//     Standard Inputs/Fix01.N22/I <-> Channel 1/Input
//     Standard Inputs/Fix01.N22/I @bit 1 <-> Channel 2/Input
//     Standard Inputs/Fix01.N22/I @bit 2 <-> Channel 3/Input
//     Standard Inputs/Fix01.N22/I @bit 3 <-> Channel 4/Input
//     Standard Inputs/Fix01.N22/I @bit 4 <-> Channel 5/Input
//     Standard Inputs/Fix01.N22/I @bit 5 <-> Channel 6/Input
//     Standard Inputs/Fix01.N22/I @bit 6 <-> Channel 7/Input
//     Standard Inputs/Fix01.N22/I @bit 7 <-> Channel 8/Input
//     Standard Inputs/Fix01.N22/InfoData/State <-> InfoData/State
//     Standard Inputs/Fix01.N22/Wc_State <-> WcState/WcState
//   SODG11_SSCC610_2403701_PLC/SODG11_SSCC610_2403701_PLC Instance <-> EtherCAT Master (EtherCAT)/IC01.T01 (EK1100)/IC01.T16 (EK1122)/Fix01.N23 (EP1008-0002)
//     Standard Inputs/Fix01.N23/I <-> Channel 1/Input
//     Standard Inputs/Fix01.N23/I @bit 1 <-> Channel 2/Input
//     Standard Inputs/Fix01.N23/I @bit 2 <-> Channel 3/Input
//     Standard Inputs/Fix01.N23/I @bit 3 <-> Channel 4/Input
//     Standard Inputs/Fix01.N23/I @bit 4 <-> Channel 5/Input
//     Standard Inputs/Fix01.N23/I @bit 5 <-> Channel 6/Input
//     Standard Inputs/Fix01.N23/I @bit 6 <-> Channel 7/Input
//     Standard Inputs/Fix01.N23/I @bit 7 <-> Channel 8/Input
//     Standard Inputs/Fix01.N23/InfoData/State <-> InfoData/State
//     Standard Inputs/Fix01.N23/Wc_State <-> WcState/WcState
//   SODG11_SSCC610_2403701_PLC/SODG11_SSCC610_2403701_PLC Instance <-> EtherCAT Master (EtherCAT)/IC01.T01 (EK1100)/IC01.T16 (EK1122)/Fix01.N24 (EP1008-0002)
//     Standard Inputs/Fix01.N24/I <-> Channel 1/Input
//     Standard Inputs/Fix01.N24/I @bit 1 <-> Channel 2/Input
//     Standard Inputs/Fix01.N24/I @bit 2 <-> Channel 3/Input
//     Standard Inputs/Fix01.N24/I @bit 3 <-> Channel 4/Input
//     Standard Inputs/Fix01.N24/I @bit 4 <-> Channel 5/Input
//     Standard Inputs/Fix01.N24/I @bit 5 <-> Channel 6/Input
//     Standard Inputs/Fix01.N24/I @bit 6 <-> Channel 7/Input
//     Standard Inputs/Fix01.N24/I @bit 7 <-> Channel 8/Input
//     Standard Inputs/Fix01.N24/InfoData/State <-> InfoData/State
//     Standard Inputs/Fix01.N24/Wc_State <-> WcState/WcState
//   SODG11_SSCC610_2403701_PLC/SODG11_SSCC610_2403701_PLC Instance <-> EtherCAT Master (EtherCAT)/IC01.T01 (EK1100)/IC01.T16 (EK1122)/Fix01.N25 (EP1008-0002)
//     Standard Inputs/Fix01.N25/I <-> Channel 1/Input
//     Standard Inputs/Fix01.N25/I @bit 1 <-> Channel 2/Input
//     Standard Inputs/Fix01.N25/I @bit 2 <-> Channel 3/Input
//     Standard Inputs/Fix01.N25/I @bit 3 <-> Channel 4/Input
//     Standard Inputs/Fix01.N25/I @bit 4 <-> Channel 5/Input
//     Standard Inputs/Fix01.N25/I @bit 5 <-> Channel 6/Input
//     Standard Inputs/Fix01.N25/I @bit 6 <-> Channel 7/Input
//     Standard Inputs/Fix01.N25/I @bit 7 <-> Channel 8/Input
//     Standard Inputs/Fix01.N25/InfoData/State <-> InfoData/State
//     Standard Inputs/Fix01.N25/Wc_State <-> WcState/WcState
//   SODG11_SSCC610_2403701_PLC/SODG11_SSCC610_2403701_PLC Instance <-> EtherCAT Master (EtherCAT)/IC01.T01 (EK1100)/IC01.T16 (EK1122)/Fix01.N26 (EP1008-0002)
//     Standard Inputs/Fix01.N26/I <-> Channel 1/Input
//     Standard Inputs/Fix01.N26/I @bit 1 <-> Channel 2/Input
//     Standard Inputs/Fix01.N26/I @bit 2 <-> Channel 3/Input
//     Standard Inputs/Fix01.N26/I @bit 3 <-> Channel 4/Input
//     Standard Inputs/Fix01.N26/I @bit 4 <-> Channel 5/Input
//     Standard Inputs/Fix01.N26/I @bit 5 <-> Channel 6/Input
//     Standard Inputs/Fix01.N26/I @bit 6 <-> Channel 7/Input
//     Standard Inputs/Fix01.N26/I @bit 7 <-> Channel 8/Input
//     Standard Inputs/Fix01.N26/InfoData/State <-> InfoData/State
//     Standard Inputs/Fix01.N26/Wc_State <-> WcState/WcState
//   SODG11_SSCC610_2403701_PLC/SODG11_SSCC610_2403701_PLC Instance <-> EtherCAT Master (EtherCAT)/IC01.T01 (EK1100)/IC01.T16 (EK1122)/Fix01.N27 (EP1008-0002)
//     Standard Inputs/Fix01.N27/I <-> Channel 1/Input
//     Standard Inputs/Fix01.N27/I @bit 1 <-> Channel 2/Input
//     Standard Inputs/Fix01.N27/I @bit 2 <-> Channel 3/Input
//     Standard Inputs/Fix01.N27/I @bit 3 <-> Channel 4/Input
//     Standard Inputs/Fix01.N27/I @bit 4 <-> Channel 5/Input
//     Standard Inputs/Fix01.N27/I @bit 5 <-> Channel 6/Input
//     Standard Inputs/Fix01.N27/I @bit 6 <-> Channel 7/Input
//     Standard Inputs/Fix01.N27/I @bit 7 <-> Channel 8/Input
//     Standard Inputs/Fix01.N27/InfoData/State <-> InfoData/State
//     Standard Inputs/Fix01.N27/Wc_State <-> WcState/WcState
//   SODG11_SSCC610_2403701_PLC/SODG11_SSCC610_2403701_PLC Instance <-> EtherCAT Master (EtherCAT)/IC01.T01 (EK1100)/IC01.T16 (EK1122)/Fix01.N28 (EP1008-0002)
//     Standard Inputs/Fix01.N28/I <-> Channel 1/Input
//     Standard Inputs/Fix01.N28/I @bit 1 <-> Channel 2/Input
//     Standard Inputs/Fix01.N28/I @bit 2 <-> Channel 3/Input
//     Standard Inputs/Fix01.N28/I @bit 3 <-> Channel 4/Input
//     Standard Inputs/Fix01.N28/I @bit 4 <-> Channel 5/Input
//     Standard Inputs/Fix01.N28/I @bit 5 <-> Channel 6/Input
//     Standard Inputs/Fix01.N28/I @bit 6 <-> Channel 7/Input
//     Standard Inputs/Fix01.N28/I @bit 7 <-> Channel 8/Input
//     Standard Inputs/Fix01.N28/InfoData/State <-> InfoData/State
//     Standard Inputs/Fix01.N28/Wc_State <-> WcState/WcState
//   SODG11_SSCC610_2403701_PLC/SODG11_SSCC610_2403701_PLC Instance <-> EtherCAT Master (EtherCAT)/IC01.T01 (EK1100)/IC01.T16 (EK1122)/Fix01.N29 (EP1008-0002)
//     Standard Inputs/Fix01.N29/I <-> Channel 1/Input
//     Standard Inputs/Fix01.N29/I @bit 1 <-> Channel 2/Input
//     Standard Inputs/Fix01.N29/I @bit 2 <-> Channel 3/Input
//     Standard Inputs/Fix01.N29/I @bit 3 <-> Channel 4/Input
//     Standard Inputs/Fix01.N29/I @bit 4 <-> Channel 5/Input
//     Standard Inputs/Fix01.N29/I @bit 5 <-> Channel 6/Input
//     Standard Inputs/Fix01.N29/I @bit 6 <-> Channel 7/Input
//     Standard Inputs/Fix01.N29/I @bit 7 <-> Channel 8/Input
//     Standard Inputs/Fix01.N29/InfoData/State <-> InfoData/State
//     Standard Inputs/Fix01.N29/Wc_State <-> WcState/WcState
//   SODG11_SSCC610_2403701_PLC/SODG11_SSCC610_2403701_PLC Instance <-> EtherCAT Master (EtherCAT)/IC01.T01 (EK1100)/IC01.T16 (EK1122)/Fix01.N30 (EP1008-0002)
//     Standard Inputs/Fix01.N30/I <-> Channel 1/Input
//     Standard Inputs/Fix01.N30/I @bit 1 <-> Channel 2/Input
//     Standard Inputs/Fix01.N30/I @bit 2 <-> Channel 3/Input
//     Standard Inputs/Fix01.N30/I @bit 3 <-> Channel 4/Input
//     Standard Inputs/Fix01.N30/I @bit 4 <-> Channel 5/Input
//     Standard Inputs/Fix01.N30/I @bit 5 <-> Channel 6/Input
//     Standard Inputs/Fix01.N30/I @bit 6 <-> Channel 7/Input
//     Standard Inputs/Fix01.N30/I @bit 7 <-> Channel 8/Input
//     Standard Inputs/Fix01.N30/InfoData/State <-> InfoData/State
//     Standard Inputs/Fix01.N30/Wc_State <-> WcState/WcState
//   SODG11_SSCC610_2403701_PLC/SODG11_SSCC610_2403701_PLC Instance <-> EtherCAT Master (EtherCAT)/IC01.T01 (EK1100)/IC01.T16 (EK1122)/Fix01.N31 (EP1008-0002)
//     Standard Inputs/Fix01.N31/I <-> Channel 1/Input
//     Standard Inputs/Fix01.N31/I @bit 1 <-> Channel 2/Input
//     Standard Inputs/Fix01.N31/I @bit 2 <-> Channel 3/Input
//     Standard Inputs/Fix01.N31/I @bit 3 <-> Channel 4/Input
//     Standard Inputs/Fix01.N31/I @bit 4 <-> Channel 5/Input
//     Standard Inputs/Fix01.N31/I @bit 5 <-> Channel 6/Input
//     Standard Inputs/Fix01.N31/I @bit 6 <-> Channel 7/Input
//     Standard Inputs/Fix01.N31/I @bit 7 <-> Channel 8/Input
//     Standard Inputs/Fix01.N31/InfoData/State <-> InfoData/State
//     Standard Inputs/Fix01.N31/Wc_State <-> WcState/WcState
//   SODG11_SSCC610_2403701_PLC/SODG11_SSCC610_2403701_PLC Instance <-> EtherCAT Master (EtherCAT)/IC01.T01 (EK1100)/IC01.T16 (EK1122)/Fix01.N90 (EP9214-0023)
//     Standard Inputs/Fix01.N90_STAT/Channel_1/Channel_Error <-> DPO Inputs Channel 1/Channel Error
//     Standard Inputs/Fix01.N90_STAT/Channel_2/Channel_Error <-> DPO Inputs Channel 2/Channel Error
//     Standard Inputs/Fix01.N90_STAT/Channel_3/Channel_Error <-> DPO Inputs Channel 3/Channel Error
//     Standard Inputs/Fix01.N90_STAT/Channel_4/Channel_Error <-> DPO Inputs Channel 4/Channel Error
//     Standard Inputs/Fix01.N90_STAT/Channel_1/Error_Up <-> DPO Inputs Channel 1/Error Up
//     Standard Inputs/Fix01.N90_STAT/Channel_2/Error_Up <-> DPO Inputs Channel 2/Error Up
//     Standard Inputs/Fix01.N90_STAT/Channel_3/Error_Up <-> DPO Inputs Channel 3/Error Up
//     Standard Inputs/Fix01.N90_STAT/Channel_4/Error_Up <-> DPO Inputs Channel 4/Error Up
//     Standard Inputs/Fix01.N90_STAT/Channel_1/Error_Us <-> DPO Inputs Channel 1/Error Us
//     Standard Inputs/Fix01.N90_STAT/Channel_2/Error_Us <-> DPO Inputs Channel 2/Error Us
//     Standard Inputs/Fix01.N90_STAT/Channel_3/Error_Us <-> DPO Inputs Channel 3/Error Us
//     Standard Inputs/Fix01.N90_STAT/Channel_4/Error_Us <-> DPO Inputs Channel 4/Error Us
//     Standard Inputs/Fix01.N90_STAT/Channel_1/Status_Up <-> DPO Inputs Channel 1/Status Up
//     Standard Inputs/Fix01.N90_STAT/Channel_2/Status_Up <-> DPO Inputs Channel 2/Status Up
//     Standard Inputs/Fix01.N90_STAT/Channel_3/Status_Up <-> DPO Inputs Channel 3/Status Up
//     Standard Inputs/Fix01.N90_STAT/Channel_4/Status_Up <-> DPO Inputs Channel 4/Status Up
//     Standard Inputs/Fix01.N90_STAT/Channel_1/Status_Us <-> DPO Inputs Channel 1/Status Us
//     Standard Inputs/Fix01.N90_STAT/Channel_2/Status_Us <-> DPO Inputs Channel 2/Status Us
//     Standard Inputs/Fix01.N90_STAT/Channel_3/Status_Us <-> DPO Inputs Channel 3/Status Us
//     Standard Inputs/Fix01.N90_STAT/Channel_4/Status_Us <-> DPO Inputs Channel 4/Status Us
//     Standard Inputs/Fix01.N90_STAT/Channel_1/SyncError <-> DPO Inputs Channel 1/Sync error
//     Standard Inputs/Fix01.N90_STAT/Channel_2/SyncError <-> DPO Inputs Channel 2/Sync error
//     Standard Inputs/Fix01.N90_STAT/Channel_3/SyncError <-> DPO Inputs Channel 3/Sync error
//     Standard Inputs/Fix01.N90_STAT/Channel_4/SyncError <-> DPO Inputs Channel 4/Sync error
//     Standard Inputs/Fix01.N90_STAT/Channel_1/TxPDO_State <-> DPO Inputs Channel 1/TxPDO State
//     Standard Inputs/Fix01.N90_STAT/Channel_2/TxPDO_State <-> DPO Inputs Channel 2/TxPDO State
//     Standard Inputs/Fix01.N90_STAT/Channel_3/TxPDO_State <-> DPO Inputs Channel 3/TxPDO State
//     Standard Inputs/Fix01.N90_STAT/Channel_4/TxPDO_State <-> DPO Inputs Channel 4/TxPDO State
//     Standard Inputs/Fix01.N90_STAT/Channel_1/TxPDO_Toggle <-> DPO Inputs Channel 1/TxPDO Toggle
//     Standard Inputs/Fix01.N90_STAT/Channel_2/TxPDO_Toggle <-> DPO Inputs Channel 2/TxPDO Toggle
//     Standard Inputs/Fix01.N90_STAT/Channel_3/TxPDO_Toggle <-> DPO Inputs Channel 3/TxPDO Toggle
//     Standard Inputs/Fix01.N90_STAT/Channel_4/TxPDO_Toggle <-> DPO Inputs Channel 4/TxPDO Toggle
//     Standard Inputs/Fix01.N90_STAT/Channel_1/Warning_Up <-> DPO Inputs Channel 1/Warning Up
//     Standard Inputs/Fix01.N90_STAT/Channel_2/Warning_Up <-> DPO Inputs Channel 2/Warning Up
//     Standard Inputs/Fix01.N90_STAT/Channel_3/Warning_Up <-> DPO Inputs Channel 3/Warning Up
//     Standard Inputs/Fix01.N90_STAT/Channel_4/Warning_Up <-> DPO Inputs Channel 4/Warning Up
//     Standard Inputs/Fix01.N90_STAT/Channel_1/Warning_Us <-> DPO Inputs Channel 1/Warning Us
//     Standard Inputs/Fix01.N90_STAT/Channel_2/Warning_Us <-> DPO Inputs Channel 2/Warning Us
//     Standard Inputs/Fix01.N90_STAT/Channel_3/Warning_Us <-> DPO Inputs Channel 3/Warning Us
//     Standard Inputs/Fix01.N90_STAT/Channel_4/Warning_Us <-> DPO Inputs Channel 4/Warning Us
//     Standard Inputs/Fix01.N90_STAT/Device/Global_Error_Bit <-> DPO Inputs Device/Global Error Bit
//     Standard Inputs/Fix01.N90_STAT/Device/Reset_Input <-> DPO Inputs Device/Reset Input
//     Standard Inputs/Fix01.N90_STAT/Device/Temperature_Error <-> DPO Inputs Device/Temperature Error
//     Standard Inputs/Fix01.N90_STAT/Device/Temperature_Warning <-> DPO Inputs Device/Temperature Warning
//     Standard Inputs/Fix01.N90_STAT/Device/TxPDO_State <-> DPO Inputs Device/TxPDO State
//     Standard Inputs/Fix01.N90_STAT/Device/TxPDO_Toggle <-> DPO Inputs Device/TxPDO Toggle
//     Standard Inputs/Fix01.N90_STAT/Device/Up_Error <-> DPO Inputs Device/Up Error
//     Standard Inputs/Fix01.N90_STAT/Device/Up_Warning <-> DPO Inputs Device/Up Warning
//     Standard Inputs/Fix01.N90_STAT/Device/Us_Error <-> DPO Inputs Device/Us Error
//     Standard Inputs/Fix01.N90_STAT/Device/Us_Warning <-> DPO Inputs Device/Us Warning
//     Standard Inputs/Fix01.N90_STAT/InfoData/AdsAddr <-> InfoData/AdsAddr
//     Standard Inputs/Fix01.N90_STAT/InfoData/State <-> InfoData/State
//     Standard Inputs/Fix01.N90_STAT/Wc_State <-> WcState/WcState
//     Standard Outputs/Fix01.N90_CMD/Channel1/Output_Up <-> DPO Outputs Channel 1/Output Up
//     Standard Outputs/Fix01.N90_CMD/Channel2/Output_Up <-> DPO Outputs Channel 2/Output Up
//     Standard Outputs/Fix01.N90_CMD/Channel3/Output_Up <-> DPO Outputs Channel 3/Output Up
//     Standard Outputs/Fix01.N90_CMD/Channel4/Output_Up <-> DPO Outputs Channel 4/Output Up
//     Standard Outputs/Fix01.N90_CMD/Channel1/Output_Us <-> DPO Outputs Channel 1/Output Us
//     Standard Outputs/Fix01.N90_CMD/Channel2/Output_Us <-> DPO Outputs Channel 2/Output Us
//     Standard Outputs/Fix01.N90_CMD/Channel3/Output_Us <-> DPO Outputs Channel 3/Output Us
//     Standard Outputs/Fix01.N90_CMD/Channel4/Output_Us <-> DPO Outputs Channel 4/Output Us
//     Standard Outputs/Fix01.N90_CMD/Channel1/Reset_Up <-> DPO Outputs Channel 1/Reset Up
//     Standard Outputs/Fix01.N90_CMD/Channel2/Reset_Up <-> DPO Outputs Channel 2/Reset Up
//     Standard Outputs/Fix01.N90_CMD/Channel3/Reset_Up <-> DPO Outputs Channel 3/Reset Up
//     Standard Outputs/Fix01.N90_CMD/Channel4/Reset_Up <-> DPO Outputs Channel 4/Reset Up
//     Standard Outputs/Fix01.N90_CMD/Channel1/Reset_Us <-> DPO Outputs Channel 1/Reset Us
//     Standard Outputs/Fix01.N90_CMD/Channel2/Reset_Us <-> DPO Outputs Channel 2/Reset Us
//     Standard Outputs/Fix01.N90_CMD/Channel3/Reset_Us <-> DPO Outputs Channel 3/Reset Us
//     Standard Outputs/Fix01.N90_CMD/Channel4/Reset_Us <-> DPO Outputs Channel 4/Reset Us
//     Standard Outputs/Fix01.N90_CMD/Device/Enable_Control_Via_Fieldbus <-> DPO Outputs Device/Enable Control Via Fieldbus
//     Standard Outputs/Fix01.N90_CMD/Device/Global_Reset <-> DPO Outputs Device/Global Reset
//   SODG11_SSCC610_2403701_PLC/SODG11_SSCC610_2403701_PLC Instance <-> EtherCAT Master (EtherCAT)/IC01.T01 (EK1100)/IC01.T16 (EK1122)/Fix01.N98  (EP2328-0002)
//     Standard Inputs/Fix01.N98.I <-> Channel 1/Input
//     Standard Inputs/Fix01.N98.I @bit 1 <-> Channel 2/Input
//     Standard Inputs/Fix01.N98.I @bit 2 <-> Channel 3/Input
//     Standard Inputs/Fix01.N98.I @bit 3 <-> Channel 4/Input
//     Standard Inputs/Fix01.N98.State <-> InfoData/State
//     Standard Inputs/Fix01.N98.WC_State <-> WcState/WcState
//     Standard Outputs/Fix01.N98.Q <-> Channel 5/Output
//     Standard Outputs/Fix01.N98.Q @bit 1 <-> Channel 6/Output
//     Standard Outputs/Fix01.N98.Q @bit 2 <-> Channel 7/Output
//     Standard Outputs/Fix01.N98.Q @bit 3 <-> Channel 8/Output
//   SODG11_SSCC610_2403701_PLC/SODG11_SSCC610_2403701_PLC Instance <-> EtherCAT Master (EtherCAT)/IC01.T01 (EK1100)/IC01.T16 (EK1122)/Fix02.N01 (EP1008-0002)
//     Standard Inputs/Fix02.N01/I <-> Channel 1/Input
//     Standard Inputs/Fix02.N01/I @bit 1 <-> Channel 2/Input
//     Standard Inputs/Fix02.N01/I @bit 2 <-> Channel 3/Input
//     Standard Inputs/Fix02.N01/I @bit 3 <-> Channel 4/Input
//     Standard Inputs/Fix02.N01/I @bit 4 <-> Channel 5/Input
//     Standard Inputs/Fix02.N01/I @bit 5 <-> Channel 6/Input
//     Standard Inputs/Fix02.N01/I @bit 6 <-> Channel 7/Input
//     Standard Inputs/Fix02.N01/I @bit 7 <-> Channel 8/Input
//     Standard Inputs/Fix02.N01/InfoData/State <-> InfoData/State
//     Standard Inputs/Fix02.N01/Wc_State <-> WcState/WcState
//   SODG11_SSCC610_2403701_PLC/SODG11_SSCC610_2403701_PLC Instance <-> EtherCAT Master (EtherCAT)/IC01.T01 (EK1100)/IC01.T16 (EK1122)/Fix02.N02 (EP1008-0002)
//     Standard Inputs/Fix02.N02/I <-> Channel 1/Input
//     Standard Inputs/Fix02.N02/I @bit 1 <-> Channel 2/Input
//     Standard Inputs/Fix02.N02/I @bit 2 <-> Channel 3/Input
//     Standard Inputs/Fix02.N02/I @bit 3 <-> Channel 4/Input
//     Standard Inputs/Fix02.N02/I @bit 4 <-> Channel 5/Input
//     Standard Inputs/Fix02.N02/I @bit 5 <-> Channel 6/Input
//     Standard Inputs/Fix02.N02/I @bit 6 <-> Channel 7/Input
//     Standard Inputs/Fix02.N02/I @bit 7 <-> Channel 8/Input
//     Standard Inputs/Fix02.N02/InfoData/State <-> InfoData/State
//     Standard Inputs/Fix02.N02/Wc_State <-> WcState/WcState
//   SODG11_SSCC610_2403701_PLC/SODG11_SSCC610_2403701_PLC Instance <-> EtherCAT Master (EtherCAT)/IC01.T01 (EK1100)/IC01.T16 (EK1122)/Fix02.N03 (EP1008-0002)
//     Standard Inputs/Fix02.N03/I <-> Channel 1/Input
//     Standard Inputs/Fix02.N03/I @bit 1 <-> Channel 2/Input
//     Standard Inputs/Fix02.N03/I @bit 2 <-> Channel 3/Input
//     Standard Inputs/Fix02.N03/I @bit 3 <-> Channel 4/Input
//     Standard Inputs/Fix02.N03/I @bit 4 <-> Channel 5/Input
//     Standard Inputs/Fix02.N03/I @bit 5 <-> Channel 6/Input
//     Standard Inputs/Fix02.N03/I @bit 6 <-> Channel 7/Input
//     Standard Inputs/Fix02.N03/I @bit 7 <-> Channel 8/Input
//     Standard Inputs/Fix02.N03/InfoData/State <-> InfoData/State
//     Standard Inputs/Fix02.N03/Wc_State <-> WcState/WcState
//   SODG11_SSCC610_2403701_PLC/SODG11_SSCC610_2403701_PLC Instance <-> EtherCAT Master (EtherCAT)/IC01.T01 (EK1100)/IC01.T16 (EK1122)/Fix02.N04 (EP1008-0002)
//     Standard Inputs/Fix02.N04/I <-> Channel 1/Input
//     Standard Inputs/Fix02.N04/I @bit 1 <-> Channel 2/Input
//     Standard Inputs/Fix02.N04/I @bit 2 <-> Channel 3/Input
//     Standard Inputs/Fix02.N04/I @bit 3 <-> Channel 4/Input
//     Standard Inputs/Fix02.N04/I @bit 4 <-> Channel 5/Input
//     Standard Inputs/Fix02.N04/I @bit 5 <-> Channel 6/Input
//     Standard Inputs/Fix02.N04/I @bit 6 <-> Channel 7/Input
//     Standard Inputs/Fix02.N04/I @bit 7 <-> Channel 8/Input
//     Standard Inputs/Fix02.N04/InfoData/State <-> InfoData/State
//     Standard Inputs/Fix02.N04/Wc_State <-> WcState/WcState
//   SODG11_SSCC610_2403701_PLC/SODG11_SSCC610_2403701_PLC Instance <-> EtherCAT Master (EtherCAT)/IC01.T01 (EK1100)/IC01.T16 (EK1122)/Fix02.N05 (EP1008-0002)
//     Standard Inputs/Fix02.N05/I <-> Channel 1/Input
//     Standard Inputs/Fix02.N05/I @bit 1 <-> Channel 2/Input
//     Standard Inputs/Fix02.N05/I @bit 2 <-> Channel 3/Input
//     Standard Inputs/Fix02.N05/I @bit 3 <-> Channel 4/Input
//     Standard Inputs/Fix02.N05/I @bit 4 <-> Channel 5/Input
//     Standard Inputs/Fix02.N05/I @bit 5 <-> Channel 6/Input
//     Standard Inputs/Fix02.N05/I @bit 6 <-> Channel 7/Input
//     Standard Inputs/Fix02.N05/I @bit 7 <-> Channel 8/Input
//     Standard Inputs/Fix02.N05/InfoData/State <-> InfoData/State
//     Standard Inputs/Fix02.N05/Wc_State <-> WcState/WcState
//   SODG11_SSCC610_2403701_PLC/SODG11_SSCC610_2403701_PLC Instance <-> EtherCAT Master (EtherCAT)/IC01.T01 (EK1100)/IC01.T16 (EK1122)/Fix02.N06 (EP1008-0002)
//     Standard Inputs/Fix02.N06/I <-> Channel 1/Input
//     Standard Inputs/Fix02.N06/I @bit 1 <-> Channel 2/Input
//     Standard Inputs/Fix02.N06/I @bit 2 <-> Channel 3/Input
//     Standard Inputs/Fix02.N06/I @bit 3 <-> Channel 4/Input
//     Standard Inputs/Fix02.N06/I @bit 4 <-> Channel 5/Input
//     Standard Inputs/Fix02.N06/I @bit 5 <-> Channel 6/Input
//     Standard Inputs/Fix02.N06/I @bit 6 <-> Channel 7/Input
//     Standard Inputs/Fix02.N06/I @bit 7 <-> Channel 8/Input
//     Standard Inputs/Fix02.N06/InfoData/State <-> InfoData/State
//     Standard Inputs/Fix02.N06/Wc_State <-> WcState/WcState
//   SODG11_SSCC610_2403701_PLC/SODG11_SSCC610_2403701_PLC Instance <-> EtherCAT Master (EtherCAT)/IC01.T01 (EK1100)/IC01.T16 (EK1122)/Fix02.N07 (EP1008-0002)
//     Standard Inputs/Fix02.N07/I <-> Channel 1/Input
//     Standard Inputs/Fix02.N07/I @bit 1 <-> Channel 2/Input
//     Standard Inputs/Fix02.N07/I @bit 2 <-> Channel 3/Input
//     Standard Inputs/Fix02.N07/I @bit 3 <-> Channel 4/Input
//     Standard Inputs/Fix02.N07/I @bit 4 <-> Channel 5/Input
//     Standard Inputs/Fix02.N07/I @bit 5 <-> Channel 6/Input
//     Standard Inputs/Fix02.N07/I @bit 6 <-> Channel 7/Input
//     Standard Inputs/Fix02.N07/I @bit 7 <-> Channel 8/Input
//     Standard Inputs/Fix02.N07/InfoData/State <-> InfoData/State
//     Standard Inputs/Fix02.N07/Wc_State <-> WcState/WcState
//   SODG11_SSCC610_2403701_PLC/SODG11_SSCC610_2403701_PLC Instance <-> EtherCAT Master (EtherCAT)/IC01.T01 (EK1100)/IC01.T16 (EK1122)/Fix02.N08 (EP1008-0002)
//     Standard Inputs/Fix02.N08/I <-> Channel 1/Input
//     Standard Inputs/Fix02.N08/I @bit 1 <-> Channel 2/Input
//     Standard Inputs/Fix02.N08/I @bit 2 <-> Channel 3/Input
//     Standard Inputs/Fix02.N08/I @bit 3 <-> Channel 4/Input
//     Standard Inputs/Fix02.N08/I @bit 4 <-> Channel 5/Input
//     Standard Inputs/Fix02.N08/I @bit 5 <-> Channel 6/Input
//     Standard Inputs/Fix02.N08/I @bit 6 <-> Channel 7/Input
//     Standard Inputs/Fix02.N08/I @bit 7 <-> Channel 8/Input
//     Standard Inputs/Fix02.N08/InfoData/State <-> InfoData/State
//     Standard Inputs/Fix02.N08/Wc_State <-> WcState/WcState
//   SODG11_SSCC610_2403701_PLC/SODG11_SSCC610_2403701_PLC Instance <-> EtherCAT Master (EtherCAT)/IC01.T01 (EK1100)/IC01.T16 (EK1122)/Fix02.N09 (EP1008-0002)
//     Standard Inputs/Fix02.N09/I <-> Channel 1/Input
//     Standard Inputs/Fix02.N09/I @bit 1 <-> Channel 2/Input
//     Standard Inputs/Fix02.N09/I @bit 2 <-> Channel 3/Input
//     Standard Inputs/Fix02.N09/I @bit 3 <-> Channel 4/Input
//     Standard Inputs/Fix02.N09/I @bit 4 <-> Channel 5/Input
//     Standard Inputs/Fix02.N09/I @bit 5 <-> Channel 6/Input
//     Standard Inputs/Fix02.N09/I @bit 6 <-> Channel 7/Input
//     Standard Inputs/Fix02.N09/I @bit 7 <-> Channel 8/Input
//     Standard Inputs/Fix02.N09/InfoData/State <-> InfoData/State
//     Standard Inputs/Fix02.N09/Wc_State <-> WcState/WcState
//   SODG11_SSCC610_2403701_PLC/SODG11_SSCC610_2403701_PLC Instance <-> EtherCAT Master (EtherCAT)/IC01.T01 (EK1100)/IC01.T16 (EK1122)/Fix02.N10 (EP1008-0002)
//     Standard Inputs/Fix02.N10/I <-> Channel 1/Input
//     Standard Inputs/Fix02.N10/I @bit 1 <-> Channel 2/Input
//     Standard Inputs/Fix02.N10/I @bit 2 <-> Channel 3/Input
//     Standard Inputs/Fix02.N10/I @bit 3 <-> Channel 4/Input
//     Standard Inputs/Fix02.N10/I @bit 4 <-> Channel 5/Input
//     Standard Inputs/Fix02.N10/I @bit 5 <-> Channel 6/Input
//     Standard Inputs/Fix02.N10/I @bit 6 <-> Channel 7/Input
//     Standard Inputs/Fix02.N10/I @bit 7 <-> Channel 8/Input
//     Standard Inputs/Fix02.N10/InfoData/State <-> InfoData/State
//     Standard Inputs/Fix02.N10/Wc_State <-> WcState/WcState
//   SODG11_SSCC610_2403701_PLC/SODG11_SSCC610_2403701_PLC Instance <-> EtherCAT Master (EtherCAT)/IC01.T01 (EK1100)/IC01.T16 (EK1122)/Fix02.N100 (EX260-SEC1)
//     Standard Inputs/Fix02.N100_STAT/InfoData/State <-> InfoData/State
//     Standard Outputs/Fix02.N100/Q <-> Byte 0/Output
//     Standard Outputs/Fix02.N100/Q @bit 8 <-> Byte 1/Output
//     Standard Outputs/Fix02.N100/Q @bit 16 <-> Byte 2/Output
//     Standard Outputs/Fix02.N100/Q @bit 24 <-> Byte 3/Output
//   SODG11_SSCC610_2403701_PLC/SODG11_SSCC610_2403701_PLC Instance <-> EtherCAT Master (EtherCAT)/IC01.T01 (EK1100)/IC01.T16 (EK1122)/Fix02.N101 (EX260-SEC1)
//     Standard Inputs/Fix02.N101_STAT/InfoData/State <-> InfoData/State
//     Standard Outputs/Fix02.N101/Q <-> Byte 0/Output
//     Standard Outputs/Fix02.N101/Q @bit 8 <-> Byte 1/Output
//     Standard Outputs/Fix02.N101/Q @bit 16 <-> Byte 2/Output
//     Standard Outputs/Fix02.N101/Q @bit 24 <-> Byte 3/Output
//   SODG11_SSCC610_2403701_PLC/SODG11_SSCC610_2403701_PLC Instance <-> EtherCAT Master (EtherCAT)/IC01.T01 (EK1100)/IC01.T16 (EK1122)/Fix02.N11 (EP1008-0002)
//     Standard Inputs/Fix02.N11/I <-> Channel 1/Input
//     Standard Inputs/Fix02.N11/I @bit 1 <-> Channel 2/Input
//     Standard Inputs/Fix02.N11/I @bit 2 <-> Channel 3/Input
//     Standard Inputs/Fix02.N11/I @bit 3 <-> Channel 4/Input
//     Standard Inputs/Fix02.N11/I @bit 4 <-> Channel 5/Input
//     Standard Inputs/Fix02.N11/I @bit 5 <-> Channel 6/Input
//     Standard Inputs/Fix02.N11/I @bit 6 <-> Channel 7/Input
//     Standard Inputs/Fix02.N11/I @bit 7 <-> Channel 8/Input
//     Standard Inputs/Fix02.N11/InfoData/State <-> InfoData/State
//     Standard Inputs/Fix02.N11/Wc_State <-> WcState/WcState
//   SODG11_SSCC610_2403701_PLC/SODG11_SSCC610_2403701_PLC Instance <-> EtherCAT Master (EtherCAT)/IC01.T01 (EK1100)/IC01.T16 (EK1122)/Fix02.N12 (EP1008-0002)
//     Standard Inputs/Fix02.N12/I <-> Channel 1/Input
//     Standard Inputs/Fix02.N12/I @bit 1 <-> Channel 2/Input
//     Standard Inputs/Fix02.N12/I @bit 2 <-> Channel 3/Input
//     Standard Inputs/Fix02.N12/I @bit 3 <-> Channel 4/Input
//     Standard Inputs/Fix02.N12/I @bit 4 <-> Channel 5/Input
//     Standard Inputs/Fix02.N12/I @bit 5 <-> Channel 6/Input
//     Standard Inputs/Fix02.N12/I @bit 6 <-> Channel 7/Input
//     Standard Inputs/Fix02.N12/I @bit 7 <-> Channel 8/Input
//     Standard Inputs/Fix02.N12/InfoData/State <-> InfoData/State
//     Standard Inputs/Fix02.N12/Wc_State <-> WcState/WcState
//   SODG11_SSCC610_2403701_PLC/SODG11_SSCC610_2403701_PLC Instance <-> EtherCAT Master (EtherCAT)/IC01.T01 (EK1100)/IC01.T16 (EK1122)/Fix02.N13 (EP1008-0002)
//     Standard Inputs/Fix02.N13/I <-> Channel 1/Input
//     Standard Inputs/Fix02.N13/I @bit 1 <-> Channel 2/Input
//     Standard Inputs/Fix02.N13/I @bit 2 <-> Channel 3/Input
//     Standard Inputs/Fix02.N13/I @bit 3 <-> Channel 4/Input
//     Standard Inputs/Fix02.N13/I @bit 4 <-> Channel 5/Input
//     Standard Inputs/Fix02.N13/I @bit 5 <-> Channel 6/Input
//     Standard Inputs/Fix02.N13/I @bit 6 <-> Channel 7/Input
//     Standard Inputs/Fix02.N13/I @bit 7 <-> Channel 8/Input
//     Standard Inputs/Fix02.N13/InfoData/State <-> InfoData/State
//     Standard Inputs/Fix02.N13/Wc_State <-> WcState/WcState
//   SODG11_SSCC610_2403701_PLC/SODG11_SSCC610_2403701_PLC Instance <-> EtherCAT Master (EtherCAT)/IC01.T01 (EK1100)/IC01.T16 (EK1122)/Fix02.N14 (EP1008-0002)
//     Standard Inputs/Fix02.N14/I <-> Channel 1/Input
//     Standard Inputs/Fix02.N14/I @bit 1 <-> Channel 2/Input
//     Standard Inputs/Fix02.N14/I @bit 2 <-> Channel 3/Input
//     Standard Inputs/Fix02.N14/I @bit 3 <-> Channel 4/Input
//     Standard Inputs/Fix02.N14/I @bit 4 <-> Channel 5/Input
//     Standard Inputs/Fix02.N14/I @bit 5 <-> Channel 6/Input
//     Standard Inputs/Fix02.N14/I @bit 6 <-> Channel 7/Input
//     Standard Inputs/Fix02.N14/I @bit 7 <-> Channel 8/Input
//     Standard Inputs/Fix02.N14/InfoData/State <-> InfoData/State
//     Standard Inputs/Fix02.N14/Wc_State <-> WcState/WcState
//   SODG11_SSCC610_2403701_PLC/SODG11_SSCC610_2403701_PLC Instance <-> EtherCAT Master (EtherCAT)/IC01.T01 (EK1100)/IC01.T16 (EK1122)/Fix02.N15 (EP1008-0002)
//     Standard Inputs/Fix02.N15/I <-> Channel 1/Input
//     Standard Inputs/Fix02.N15/I @bit 1 <-> Channel 2/Input
//     Standard Inputs/Fix02.N15/I @bit 2 <-> Channel 3/Input
//     Standard Inputs/Fix02.N15/I @bit 3 <-> Channel 4/Input
//     Standard Inputs/Fix02.N15/I @bit 4 <-> Channel 5/Input
//     Standard Inputs/Fix02.N15/I @bit 5 <-> Channel 6/Input
//     Standard Inputs/Fix02.N15/I @bit 6 <-> Channel 7/Input
//     Standard Inputs/Fix02.N15/I @bit 7 <-> Channel 8/Input
//     Standard Inputs/Fix02.N15/InfoData/State <-> InfoData/State
//     Standard Inputs/Fix02.N15/Wc_State <-> WcState/WcState
//   SODG11_SSCC610_2403701_PLC/SODG11_SSCC610_2403701_PLC Instance <-> EtherCAT Master (EtherCAT)/IC01.T01 (EK1100)/IC01.T16 (EK1122)/Fix02.N16 (EP1008-0002)
//     Standard Inputs/Fix02.N16/I <-> Channel 1/Input
//     Standard Inputs/Fix02.N16/I @bit 1 <-> Channel 2/Input
//     Standard Inputs/Fix02.N16/I @bit 2 <-> Channel 3/Input
//     Standard Inputs/Fix02.N16/I @bit 3 <-> Channel 4/Input
//     Standard Inputs/Fix02.N16/I @bit 4 <-> Channel 5/Input
//     Standard Inputs/Fix02.N16/I @bit 5 <-> Channel 6/Input
//     Standard Inputs/Fix02.N16/I @bit 6 <-> Channel 7/Input
//     Standard Inputs/Fix02.N16/I @bit 7 <-> Channel 8/Input
//     Standard Inputs/Fix02.N16/InfoData/State <-> InfoData/State
//     Standard Inputs/Fix02.N16/Wc_State <-> WcState/WcState
//   SODG11_SSCC610_2403701_PLC/SODG11_SSCC610_2403701_PLC Instance <-> EtherCAT Master (EtherCAT)/IC01.T01 (EK1100)/IC01.T16 (EK1122)/Fix02.N17 (EP1008-0002)
//     Standard Inputs/Fix02.N17/I <-> Channel 1/Input
//     Standard Inputs/Fix02.N17/I @bit 1 <-> Channel 2/Input
//     Standard Inputs/Fix02.N17/I @bit 2 <-> Channel 3/Input
//     Standard Inputs/Fix02.N17/I @bit 3 <-> Channel 4/Input
//     Standard Inputs/Fix02.N17/I @bit 4 <-> Channel 5/Input
//     Standard Inputs/Fix02.N17/I @bit 5 <-> Channel 6/Input
//     Standard Inputs/Fix02.N17/I @bit 6 <-> Channel 7/Input
//     Standard Inputs/Fix02.N17/I @bit 7 <-> Channel 8/Input
//     Standard Inputs/Fix02.N17/InfoData/State <-> InfoData/State
//     Standard Inputs/Fix02.N17/Wc_State <-> WcState/WcState
//   SODG11_SSCC610_2403701_PLC/SODG11_SSCC610_2403701_PLC Instance <-> EtherCAT Master (EtherCAT)/IC01.T01 (EK1100)/IC01.T16 (EK1122)/Fix02.N18 (EP1008-0002)
//     Standard Inputs/Fix02.N18/I <-> Channel 1/Input
//     Standard Inputs/Fix02.N18/I @bit 1 <-> Channel 2/Input
//     Standard Inputs/Fix02.N18/I @bit 2 <-> Channel 3/Input
//     Standard Inputs/Fix02.N18/I @bit 3 <-> Channel 4/Input
//     Standard Inputs/Fix02.N18/I @bit 4 <-> Channel 5/Input
//     Standard Inputs/Fix02.N18/I @bit 5 <-> Channel 6/Input
//     Standard Inputs/Fix02.N18/I @bit 6 <-> Channel 7/Input
//     Standard Inputs/Fix02.N18/I @bit 7 <-> Channel 8/Input
//     Standard Inputs/Fix02.N18/InfoData/State <-> InfoData/State
//     Standard Inputs/Fix02.N18/Wc_State <-> WcState/WcState
//   SODG11_SSCC610_2403701_PLC/SODG11_SSCC610_2403701_PLC Instance <-> EtherCAT Master (EtherCAT)/IC01.T01 (EK1100)/IC01.T16 (EK1122)/Fix02.N19 (EP1008-0002)
//     Standard Inputs/Fix02.N19/I <-> Channel 1/Input
//     Standard Inputs/Fix02.N19/I @bit 1 <-> Channel 2/Input
//     Standard Inputs/Fix02.N19/I @bit 2 <-> Channel 3/Input
//     Standard Inputs/Fix02.N19/I @bit 3 <-> Channel 4/Input
//     Standard Inputs/Fix02.N19/I @bit 4 <-> Channel 5/Input
//     Standard Inputs/Fix02.N19/I @bit 5 <-> Channel 6/Input
//     Standard Inputs/Fix02.N19/I @bit 6 <-> Channel 7/Input
//     Standard Inputs/Fix02.N19/I @bit 7 <-> Channel 8/Input
//     Standard Inputs/Fix02.N19/InfoData/State <-> InfoData/State
//     Standard Inputs/Fix02.N19/Wc_State <-> WcState/WcState
//   SODG11_SSCC610_2403701_PLC/SODG11_SSCC610_2403701_PLC Instance <-> EtherCAT Master (EtherCAT)/IC01.T01 (EK1100)/IC01.T16 (EK1122)/Fix02.N20 (EP1008-0002)
//     Standard Inputs/Fix02.N20/I <-> Channel 1/Input
//     Standard Inputs/Fix02.N20/I @bit 1 <-> Channel 2/Input
//     Standard Inputs/Fix02.N20/I @bit 2 <-> Channel 3/Input
//     Standard Inputs/Fix02.N20/I @bit 3 <-> Channel 4/Input
//     Standard Inputs/Fix02.N20/I @bit 4 <-> Channel 5/Input
//     Standard Inputs/Fix02.N20/I @bit 5 <-> Channel 6/Input
//     Standard Inputs/Fix02.N20/I @bit 6 <-> Channel 7/Input
//     Standard Inputs/Fix02.N20/I @bit 7 <-> Channel 8/Input
//     Standard Inputs/Fix02.N20/InfoData/State <-> InfoData/State
//     Standard Inputs/Fix02.N20/Wc_State <-> WcState/WcState
//   SODG11_SSCC610_2403701_PLC/SODG11_SSCC610_2403701_PLC Instance <-> EtherCAT Master (EtherCAT)/IC01.T01 (EK1100)/IC01.T16 (EK1122)/Fix02.N21 (EP1008-0002)
//     Standard Inputs/Fix02.N21/I <-> Channel 1/Input
//     Standard Inputs/Fix02.N21/I @bit 1 <-> Channel 2/Input
//     Standard Inputs/Fix02.N21/I @bit 2 <-> Channel 3/Input
//     Standard Inputs/Fix02.N21/I @bit 3 <-> Channel 4/Input
//     Standard Inputs/Fix02.N21/I @bit 4 <-> Channel 5/Input
//     Standard Inputs/Fix02.N21/I @bit 5 <-> Channel 6/Input
//     Standard Inputs/Fix02.N21/I @bit 6 <-> Channel 7/Input
//     Standard Inputs/Fix02.N21/I @bit 7 <-> Channel 8/Input
//     Standard Inputs/Fix02.N21/InfoData/State <-> InfoData/State
//     Standard Inputs/Fix02.N21/Wc_State <-> WcState/WcState
//   SODG11_SSCC610_2403701_PLC/SODG11_SSCC610_2403701_PLC Instance <-> EtherCAT Master (EtherCAT)/IC01.T01 (EK1100)/IC01.T16 (EK1122)/Fix02.N22 (EP1008-0002)
//     Standard Inputs/Fix02.N22/I <-> Channel 1/Input
//     Standard Inputs/Fix02.N22/I @bit 1 <-> Channel 2/Input
//     Standard Inputs/Fix02.N22/I @bit 2 <-> Channel 3/Input
//     Standard Inputs/Fix02.N22/I @bit 3 <-> Channel 4/Input
//     Standard Inputs/Fix02.N22/I @bit 4 <-> Channel 5/Input
//     Standard Inputs/Fix02.N22/I @bit 5 <-> Channel 6/Input
//     Standard Inputs/Fix02.N22/I @bit 6 <-> Channel 7/Input
//     Standard Inputs/Fix02.N22/I @bit 7 <-> Channel 8/Input
//     Standard Inputs/Fix02.N22/InfoData/State <-> InfoData/State
//     Standard Inputs/Fix02.N22/Wc_State <-> WcState/WcState
//   SODG11_SSCC610_2403701_PLC/SODG11_SSCC610_2403701_PLC Instance <-> EtherCAT Master (EtherCAT)/IC01.T01 (EK1100)/IC01.T16 (EK1122)/Fix02.N23 (EP1008-0002)
//     Standard Inputs/Fix02.N23/I <-> Channel 1/Input
//     Standard Inputs/Fix02.N23/I @bit 1 <-> Channel 2/Input
//     Standard Inputs/Fix02.N23/I @bit 2 <-> Channel 3/Input
//     Standard Inputs/Fix02.N23/I @bit 3 <-> Channel 4/Input
//     Standard Inputs/Fix02.N23/I @bit 4 <-> Channel 5/Input
//     Standard Inputs/Fix02.N23/I @bit 5 <-> Channel 6/Input
//     Standard Inputs/Fix02.N23/I @bit 6 <-> Channel 7/Input
//     Standard Inputs/Fix02.N23/I @bit 7 <-> Channel 8/Input
//     Standard Inputs/Fix02.N23/InfoData/State <-> InfoData/State
//     Standard Inputs/Fix02.N23/Wc_State <-> WcState/WcState
//   SODG11_SSCC610_2403701_PLC/SODG11_SSCC610_2403701_PLC Instance <-> EtherCAT Master (EtherCAT)/IC01.T01 (EK1100)/IC01.T16 (EK1122)/Fix02.N24 (EP1008-0002)
//     Standard Inputs/Fix02.N24/I <-> Channel 1/Input
//     Standard Inputs/Fix02.N24/I @bit 1 <-> Channel 2/Input
//     Standard Inputs/Fix02.N24/I @bit 2 <-> Channel 3/Input
//     Standard Inputs/Fix02.N24/I @bit 3 <-> Channel 4/Input
//     Standard Inputs/Fix02.N24/I @bit 4 <-> Channel 5/Input
//     Standard Inputs/Fix02.N24/I @bit 5 <-> Channel 6/Input
//     Standard Inputs/Fix02.N24/I @bit 6 <-> Channel 7/Input
//     Standard Inputs/Fix02.N24/I @bit 7 <-> Channel 8/Input
//     Standard Inputs/Fix02.N24/InfoData/State <-> InfoData/State
//     Standard Inputs/Fix02.N24/Wc_State <-> WcState/WcState
//   SODG11_SSCC610_2403701_PLC/SODG11_SSCC610_2403701_PLC Instance <-> EtherCAT Master (EtherCAT)/IC01.T01 (EK1100)/IC01.T16 (EK1122)/Fix02.N25 (EP1008-0002)
//     Standard Inputs/Fix02.N25/I <-> Channel 1/Input
//     Standard Inputs/Fix02.N25/I @bit 1 <-> Channel 2/Input
//     Standard Inputs/Fix02.N25/I @bit 2 <-> Channel 3/Input
//     Standard Inputs/Fix02.N25/I @bit 3 <-> Channel 4/Input
//     Standard Inputs/Fix02.N25/I @bit 4 <-> Channel 5/Input
//     Standard Inputs/Fix02.N25/I @bit 5 <-> Channel 6/Input
//     Standard Inputs/Fix02.N25/I @bit 6 <-> Channel 7/Input
//     Standard Inputs/Fix02.N25/I @bit 7 <-> Channel 8/Input
//     Standard Inputs/Fix02.N25/InfoData/State <-> InfoData/State
//     Standard Inputs/Fix02.N25/Wc_State <-> WcState/WcState
//   SODG11_SSCC610_2403701_PLC/SODG11_SSCC610_2403701_PLC Instance <-> EtherCAT Master (EtherCAT)/IC01.T01 (EK1100)/IC01.T16 (EK1122)/Fix02.N26 (EP1008-0002)
//     Standard Inputs/Fix02.N26/I <-> Channel 1/Input
//     Standard Inputs/Fix02.N26/I @bit 1 <-> Channel 2/Input
//     Standard Inputs/Fix02.N26/I @bit 2 <-> Channel 3/Input
//     Standard Inputs/Fix02.N26/I @bit 3 <-> Channel 4/Input
//     Standard Inputs/Fix02.N26/I @bit 4 <-> Channel 5/Input
//     Standard Inputs/Fix02.N26/I @bit 5 <-> Channel 6/Input
//     Standard Inputs/Fix02.N26/I @bit 6 <-> Channel 7/Input
//     Standard Inputs/Fix02.N26/I @bit 7 <-> Channel 8/Input
//     Standard Inputs/Fix02.N26/InfoData/State <-> InfoData/State
//     Standard Inputs/Fix02.N26/Wc_State <-> WcState/WcState
//   SODG11_SSCC610_2403701_PLC/SODG11_SSCC610_2403701_PLC Instance <-> EtherCAT Master (EtherCAT)/IC01.T01 (EK1100)/IC01.T16 (EK1122)/Fix02.N27 (EP1008-0002)
//     Standard Inputs/Fix02.N27/I <-> Channel 1/Input
//     Standard Inputs/Fix02.N27/I @bit 1 <-> Channel 2/Input
//     Standard Inputs/Fix02.N27/I @bit 2 <-> Channel 3/Input
//     Standard Inputs/Fix02.N27/I @bit 3 <-> Channel 4/Input
//     Standard Inputs/Fix02.N27/I @bit 4 <-> Channel 5/Input
//     Standard Inputs/Fix02.N27/I @bit 5 <-> Channel 6/Input
//     Standard Inputs/Fix02.N27/I @bit 6 <-> Channel 7/Input
//     Standard Inputs/Fix02.N27/I @bit 7 <-> Channel 8/Input
//     Standard Inputs/Fix02.N27/InfoData/State <-> InfoData/State
//     Standard Inputs/Fix02.N27/Wc_State <-> WcState/WcState
//   SODG11_SSCC610_2403701_PLC/SODG11_SSCC610_2403701_PLC Instance <-> EtherCAT Master (EtherCAT)/IC01.T01 (EK1100)/IC01.T16 (EK1122)/Fix02.N28(EP1008-0002)
//     Standard Inputs/Fix02.N28/I <-> Channel 1/Input
//     Standard Inputs/Fix02.N28/I @bit 1 <-> Channel 2/Input
//     Standard Inputs/Fix02.N28/I @bit 2 <-> Channel 3/Input
//     Standard Inputs/Fix02.N28/I @bit 3 <-> Channel 4/Input
//     Standard Inputs/Fix02.N28/I @bit 4 <-> Channel 5/Input
//     Standard Inputs/Fix02.N28/I @bit 5 <-> Channel 6/Input
//     Standard Inputs/Fix02.N28/I @bit 6 <-> Channel 7/Input
//     Standard Inputs/Fix02.N28/I @bit 7 <-> Channel 8/Input
//     Standard Inputs/Fix02.N28/InfoData/State <-> InfoData/State
//     Standard Inputs/Fix02.N28/Wc_State <-> WcState/WcState
//   SODG11_SSCC610_2403701_PLC/SODG11_SSCC610_2403701_PLC Instance <-> EtherCAT Master (EtherCAT)/IC01.T01 (EK1100)/IC01.T16 (EK1122)/Fix02.N29 (EP1008-0002)
//     Standard Inputs/Fix02.N29/I <-> Channel 1/Input
//     Standard Inputs/Fix02.N29/I @bit 1 <-> Channel 2/Input
//     Standard Inputs/Fix02.N29/I @bit 2 <-> Channel 3/Input
//     Standard Inputs/Fix02.N29/I @bit 3 <-> Channel 4/Input
//     Standard Inputs/Fix02.N29/I @bit 4 <-> Channel 5/Input
//     Standard Inputs/Fix02.N29/I @bit 5 <-> Channel 6/Input
//     Standard Inputs/Fix02.N29/I @bit 6 <-> Channel 7/Input
//     Standard Inputs/Fix02.N29/I @bit 7 <-> Channel 8/Input
//     Standard Inputs/Fix02.N29/InfoData/State <-> InfoData/State
//     Standard Inputs/Fix02.N29/Wc_State <-> WcState/WcState
//   SODG11_SSCC610_2403701_PLC/SODG11_SSCC610_2403701_PLC Instance <-> EtherCAT Master (EtherCAT)/IC01.T01 (EK1100)/IC01.T16 (EK1122)/Fix02.N30 (EP1008-0002)
//     Standard Inputs/Fix02.N30/I <-> Channel 1/Input
//     Standard Inputs/Fix02.N30/I @bit 1 <-> Channel 2/Input
//     Standard Inputs/Fix02.N30/I @bit 2 <-> Channel 3/Input
//     Standard Inputs/Fix02.N30/I @bit 3 <-> Channel 4/Input
//     Standard Inputs/Fix02.N30/I @bit 4 <-> Channel 5/Input
//     Standard Inputs/Fix02.N30/I @bit 5 <-> Channel 6/Input
//     Standard Inputs/Fix02.N30/I @bit 6 <-> Channel 7/Input
//     Standard Inputs/Fix02.N30/I @bit 7 <-> Channel 8/Input
//     Standard Inputs/Fix02.N30/InfoData/State <-> InfoData/State
//     Standard Inputs/Fix02.N30/Wc_State <-> WcState/WcState
//   SODG11_SSCC610_2403701_PLC/SODG11_SSCC610_2403701_PLC Instance <-> EtherCAT Master (EtherCAT)/IC01.T01 (EK1100)/IC01.T16 (EK1122)/Fix02.N31 (EP1008-0002)
//     Standard Inputs/Fix02.N31/I <-> Channel 1/Input
//     Standard Inputs/Fix02.N31/I @bit 1 <-> Channel 2/Input
//     Standard Inputs/Fix02.N31/I @bit 2 <-> Channel 3/Input
//     Standard Inputs/Fix02.N31/I @bit 3 <-> Channel 4/Input
//     Standard Inputs/Fix02.N31/I @bit 4 <-> Channel 5/Input
//     Standard Inputs/Fix02.N31/I @bit 5 <-> Channel 6/Input
//     Standard Inputs/Fix02.N31/I @bit 6 <-> Channel 7/Input
//     Standard Inputs/Fix02.N31/I @bit 7 <-> Channel 8/Input
//     Standard Inputs/Fix02.N31/InfoData/State <-> InfoData/State
//     Standard Inputs/Fix02.N31/Wc_State <-> WcState/WcState
//   SODG11_SSCC610_2403701_PLC/SODG11_SSCC610_2403701_PLC Instance <-> EtherCAT Master (EtherCAT)/IC01.T01 (EK1100)/IC01.T16 (EK1122)/Fix02.N90 (EP9214-0023)
//     Standard Inputs/Fix02.N90_STAT/Channel_1/Channel_Error <-> DPO Inputs Channel 1/Channel Error
//     Standard Inputs/Fix02.N90_STAT/Channel_2/Channel_Error <-> DPO Inputs Channel 2/Channel Error
//     Standard Inputs/Fix02.N90_STAT/Channel_3/Channel_Error <-> DPO Inputs Channel 3/Channel Error
//     Standard Inputs/Fix02.N90_STAT/Channel_4/Channel_Error <-> DPO Inputs Channel 4/Channel Error
//     Standard Inputs/Fix02.N90_STAT/Channel_1/Error_Up <-> DPO Inputs Channel 1/Error Up
//     Standard Inputs/Fix02.N90_STAT/Channel_2/Error_Up <-> DPO Inputs Channel 2/Error Up
//     Standard Inputs/Fix02.N90_STAT/Channel_3/Error_Up <-> DPO Inputs Channel 3/Error Up
//     Standard Inputs/Fix02.N90_STAT/Channel_4/Error_Up <-> DPO Inputs Channel 4/Error Up
//     Standard Inputs/Fix02.N90_STAT/Channel_1/Error_Us <-> DPO Inputs Channel 1/Error Us
//     Standard Inputs/Fix02.N90_STAT/Channel_2/Error_Us <-> DPO Inputs Channel 2/Error Us
//     Standard Inputs/Fix02.N90_STAT/Channel_3/Error_Us <-> DPO Inputs Channel 3/Error Us
//     Standard Inputs/Fix02.N90_STAT/Channel_4/Error_Us <-> DPO Inputs Channel 4/Error Us
//     Standard Inputs/Fix02.N90_STAT/Channel_1/Status_Up <-> DPO Inputs Channel 1/Status Up
//     Standard Inputs/Fix02.N90_STAT/Channel_2/Status_Up <-> DPO Inputs Channel 2/Status Up
//     Standard Inputs/Fix02.N90_STAT/Channel_3/Status_Up <-> DPO Inputs Channel 3/Status Up
//     Standard Inputs/Fix02.N90_STAT/Channel_4/Status_Up <-> DPO Inputs Channel 4/Status Up
//     Standard Inputs/Fix02.N90_STAT/Channel_1/Status_Us <-> DPO Inputs Channel 1/Status Us
//     Standard Inputs/Fix02.N90_STAT/Channel_2/Status_Us <-> DPO Inputs Channel 2/Status Us
//     Standard Inputs/Fix02.N90_STAT/Channel_3/Status_Us <-> DPO Inputs Channel 3/Status Us
//     Standard Inputs/Fix02.N90_STAT/Channel_4/Status_Us <-> DPO Inputs Channel 4/Status Us
//     Standard Inputs/Fix02.N90_STAT/Channel_1/SyncError <-> DPO Inputs Channel 1/Sync error
//     Standard Inputs/Fix02.N90_STAT/Channel_2/SyncError <-> DPO Inputs Channel 2/Sync error
//     Standard Inputs/Fix02.N90_STAT/Channel_3/SyncError <-> DPO Inputs Channel 3/Sync error
//     Standard Inputs/Fix02.N90_STAT/Channel_4/SyncError <-> DPO Inputs Channel 4/Sync error
//     Standard Inputs/Fix02.N90_STAT/Channel_1/TxPDO_State <-> DPO Inputs Channel 1/TxPDO State
//     Standard Inputs/Fix02.N90_STAT/Channel_2/TxPDO_State <-> DPO Inputs Channel 2/TxPDO State
//     Standard Inputs/Fix02.N90_STAT/Channel_3/TxPDO_State <-> DPO Inputs Channel 3/TxPDO State
//     Standard Inputs/Fix02.N90_STAT/Channel_4/TxPDO_State <-> DPO Inputs Channel 4/TxPDO State
//     Standard Inputs/Fix02.N90_STAT/Channel_1/TxPDO_Toggle <-> DPO Inputs Channel 1/TxPDO Toggle
//     Standard Inputs/Fix02.N90_STAT/Channel_2/TxPDO_Toggle <-> DPO Inputs Channel 2/TxPDO Toggle
//     Standard Inputs/Fix02.N90_STAT/Channel_3/TxPDO_Toggle <-> DPO Inputs Channel 3/TxPDO Toggle
//     Standard Inputs/Fix02.N90_STAT/Channel_4/TxPDO_Toggle <-> DPO Inputs Channel 4/TxPDO Toggle
//     Standard Inputs/Fix02.N90_STAT/Channel_1/Warning_Up <-> DPO Inputs Channel 1/Warning Up
//     Standard Inputs/Fix02.N90_STAT/Channel_2/Warning_Up <-> DPO Inputs Channel 2/Warning Up
//     Standard Inputs/Fix02.N90_STAT/Channel_3/Warning_Up <-> DPO Inputs Channel 3/Warning Up
//     Standard Inputs/Fix02.N90_STAT/Channel_4/Warning_Up <-> DPO Inputs Channel 4/Warning Up
//     Standard Inputs/Fix02.N90_STAT/Channel_1/Warning_Us <-> DPO Inputs Channel 1/Warning Us
//     Standard Inputs/Fix02.N90_STAT/Channel_2/Warning_Us <-> DPO Inputs Channel 2/Warning Us
//     Standard Inputs/Fix02.N90_STAT/Channel_3/Warning_Us <-> DPO Inputs Channel 3/Warning Us
//     Standard Inputs/Fix02.N90_STAT/Channel_4/Warning_Us <-> DPO Inputs Channel 4/Warning Us
//     Standard Inputs/Fix02.N90_STAT/Device/Global_Error_Bit <-> DPO Inputs Device/Global Error Bit
//     Standard Inputs/Fix02.N90_STAT/Device/Reset_Input <-> DPO Inputs Device/Reset Input
//     Standard Inputs/Fix02.N90_STAT/Device/Temperature_Error <-> DPO Inputs Device/Temperature Error
//     Standard Inputs/Fix02.N90_STAT/Device/Temperature_Warning <-> DPO Inputs Device/Temperature Warning
//     Standard Inputs/Fix02.N90_STAT/Device/TxPDO_State <-> DPO Inputs Device/TxPDO State
//     Standard Inputs/Fix02.N90_STAT/Device/TxPDO_Toggle <-> DPO Inputs Device/TxPDO Toggle
//     Standard Inputs/Fix02.N90_STAT/Device/Up_Error <-> DPO Inputs Device/Up Error
//     Standard Inputs/Fix02.N90_STAT/Device/Up_Warning <-> DPO Inputs Device/Up Warning
//     Standard Inputs/Fix02.N90_STAT/Device/Us_Error <-> DPO Inputs Device/Us Error
//     Standard Inputs/Fix02.N90_STAT/Device/Us_Warning <-> DPO Inputs Device/Us Warning
//     Standard Inputs/Fix02.N90_STAT/InfoData/AdsAddr <-> InfoData/AdsAddr
//     Standard Inputs/Fix02.N90_STAT/InfoData/State <-> InfoData/State
//     Standard Inputs/Fix02.N90_STAT/Wc_State <-> WcState/WcState
//     Standard Outputs/Fix02.N90_CMD/Channel1/Output_Up <-> DPO Outputs Channel 1/Output Up
//     Standard Outputs/Fix02.N90_CMD/Channel2/Output_Up <-> DPO Outputs Channel 2/Output Up
//     Standard Outputs/Fix02.N90_CMD/Channel3/Output_Up <-> DPO Outputs Channel 3/Output Up
//     Standard Outputs/Fix02.N90_CMD/Channel4/Output_Up <-> DPO Outputs Channel 4/Output Up
//     Standard Outputs/Fix02.N90_CMD/Channel1/Output_Us <-> DPO Outputs Channel 1/Output Us
//     Standard Outputs/Fix02.N90_CMD/Channel2/Output_Us <-> DPO Outputs Channel 2/Output Us
//     Standard Outputs/Fix02.N90_CMD/Channel3/Output_Us <-> DPO Outputs Channel 3/Output Us
//     Standard Outputs/Fix02.N90_CMD/Channel4/Output_Us <-> DPO Outputs Channel 4/Output Us
//     Standard Outputs/Fix02.N90_CMD/Channel1/Reset_Up <-> DPO Outputs Channel 1/Reset Up
//     Standard Outputs/Fix02.N90_CMD/Channel2/Reset_Up <-> DPO Outputs Channel 2/Reset Up
//     Standard Outputs/Fix02.N90_CMD/Channel3/Reset_Up <-> DPO Outputs Channel 3/Reset Up
//     Standard Outputs/Fix02.N90_CMD/Channel4/Reset_Up <-> DPO Outputs Channel 4/Reset Up
//     Standard Outputs/Fix02.N90_CMD/Channel1/Reset_Us <-> DPO Outputs Channel 1/Reset Us
//     Standard Outputs/Fix02.N90_CMD/Channel2/Reset_Us <-> DPO Outputs Channel 2/Reset Us
//     Standard Outputs/Fix02.N90_CMD/Channel3/Reset_Us <-> DPO Outputs Channel 3/Reset Us
//     Standard Outputs/Fix02.N90_CMD/Channel4/Reset_Us <-> DPO Outputs Channel 4/Reset Us
//     Standard Outputs/Fix02.N90_CMD/Device/Enable_Control_Via_Fieldbus <-> DPO Outputs Device/Enable Control Via Fieldbus
//     Standard Outputs/Fix02.N90_CMD/Device/Global_Reset <-> DPO Outputs Device/Global Reset
//   SODG11_SSCC610_2403701_PLC/SODG11_SSCC610_2403701_PLC Instance <-> EtherCAT Master (EtherCAT)/IC01.T01 (EK1100)/IC01.T16 (EK1122)/Fix02.N98(EP2328-0002)
//     Standard Inputs/Fix02.N98.I <-> Channel 1/Input
//     Standard Inputs/Fix02.N98.I @bit 1 <-> Channel 2/Input
//     Standard Inputs/Fix02.N98.I @bit 2 <-> Channel 3/Input
//     Standard Inputs/Fix02.N98.I @bit 3 <-> Channel 4/Input
//     Standard Inputs/Fix02.N98.State <-> InfoData/State
//     Standard Inputs/Fix02.N98.WC_State <-> WcState/WcState
//     Standard Outputs/Fix02.N98.Q <-> Channel 5/Output
//     Standard Outputs/Fix02.N98.Q @bit 1 <-> Channel 6/Output
//     Standard Outputs/Fix02.N98.Q @bit 2 <-> Channel 7/Output
//     Standard Outputs/Fix02.N98.Q @bit 3 <-> Channel 8/Output
//   SODG11_SSCC610_2403701_PLC/SODG11_SSCC610_2403701_PLC Instance <-> EtherCAT Master (EtherCAT)/IC02.T01 (EK1100)
//     Standard Inputs/MAIN.IC02.T01/InfoData/State <-> InfoData/State
//   SODG11_SSCC610_2403701_PLC/SODG11_SSCC610_2403701_PLC Instance <-> EtherCAT Master (EtherCAT)/IC02.T01 (EK1100)/IC02.T02 (EL6900)
//     Standard Inputs/MAIN.Access_Violation_IC02 <-> StandardInputs/Standard Out Var 30
//     Standard Inputs/MAIN.IC02.T02_STAT/Device_Info_Data/Project_CRC <-> Device Info Data/Project CRC
//     Standard Inputs/MAIN.IC02.T02_STAT/FBs_FB_ERR <-> StandardInputs/Standard Out Var 26
//     Standard Inputs/MAIN.IC02.T02_STAT/FBs_FB_ERR @bit 8 <-> StandardInputs/Standard Out Var 27
//     Standard Inputs/MAIN.IC02.T02_STAT/FBs_FB_ERR @bit 17 <-> StandardInputs/Standard Out Var 28
//     Standard Inputs/MAIN.IC02.T02_STAT/FBs_FB_ERR @bit 16 <-> StandardInputs/Standard Out Var 29
//     Standard Inputs/MAIN.IC02.T02_STAT/InfoData/AdsAddr/netId <-> InfoData/AdsAddr/netId
//     Standard Inputs/MAIN.IC02.T02_STAT/InfoData/AdsAddr/port <-> InfoData/AdsAddr/port
//     Standard Inputs/MAIN.IC02.T02_STAT/InfoData/State <-> InfoData/State
//     Standard Inputs/MAIN.IC02.T02_STAT/SGs_COM_ERR <-> StandardInputs/Standard Out Var 17
//     Standard Inputs/MAIN.IC02.T02_STAT/SGs_COM_ERR @bit 1 <-> StandardInputs/Standard Out Var 20
//     Standard Inputs/MAIN.IC02.T02_STAT/SGs_FB_ERR <-> StandardInputs/Standard Out Var 16
//     Standard Inputs/MAIN.IC02.T02_STAT/SGs_FB_ERR @bit 1 <-> StandardInputs/Standard Out Var 19
//     Standard Inputs/MAIN.IC02.T02_STAT/SGs_OUT_ERR <-> StandardInputs/Standard Out Var 18
//     Standard Inputs/MAIN.IC02.T02_STAT/SGs_OUT_ERR @bit 1 <-> StandardInputs/Standard Out Var 25
//     Standard Inputs/MAIN.IC02.T09/Q <-> StandardInputs/Standard Out Var 21
//     Standard Inputs/MAIN.IC02.T10/Q <-> StandardInputs/Standard Out Var 23
//     Standard Inputs/MAIN.IC02.T09/Q @bit 1 <-> StandardInputs/Standard Out Var 22
//     Standard Inputs/MAIN.IC02.T10/Q @bit 1 <-> StandardInputs/Standard Out Var 24
//     Standard Outputs/MAIN.IC02.T02_CMD/FBs_ControlPowerPB <-> StandardOutputs/Standard In Var 14
//     Standard Outputs/MAIN.IC02.T02_CMD/SGs_ERRAck <-> StandardOutputs/Standard In Var 11
//     Standard Outputs/MAIN.IC02.T02_CMD/SGs_ERRAck <-> StandardOutputs/Standard In Var 13
//     Standard Outputs/MAIN.IC02.T02_CMD/SGs_RUNSTOP <-> StandardOutputs/Standard In Var 10
//     Standard Outputs/MAIN.IC02.T02_CMD/SGs_RUNSTOP <-> StandardOutputs/Standard In Var 12
//   SODG11_SSCC610_2403701_PLC/SODG11_SSCC610_2403701_PLC Instance <-> EtherCAT Master (EtherCAT)/IC02.T01 (EK1100)/IC02.T03 (EL1904)
//     Standard Inputs/MAIN.IC02.T03/I <-> Module 1 (FSOES)/TxPDO/FSOE/InputChannel1
//     Standard Inputs/MAIN.IC02.T03/I @bit 1 <-> Module 1 (FSOES)/TxPDO/FSOE/InputChannel2
//     Standard Inputs/MAIN.IC02.T03/I @bit 2 <-> Module 1 (FSOES)/TxPDO/FSOE/InputChannel3
//     Standard Inputs/MAIN.IC02.T03/I @bit 3 <-> Module 1 (FSOES)/TxPDO/FSOE/InputChannel4
//     Standard Inputs/MAIN.IC02.T03/InfoData/State <-> InfoData/State
//   SODG11_SSCC610_2403701_PLC/SODG11_SSCC610_2403701_PLC Instance <-> EtherCAT Master (EtherCAT)/IC02.T01 (EK1100)/IC02.T04 (EL1904)
//     Standard Inputs/MAIN.IC02.T04/I <-> Module 1 (FSOES)/TxPDO/FSOE/InputChannel1
//     Standard Inputs/MAIN.IC02.T04/I @bit 1 <-> Module 1 (FSOES)/TxPDO/FSOE/InputChannel2
//     Standard Inputs/MAIN.IC02.T04/I @bit 2 <-> Module 1 (FSOES)/TxPDO/FSOE/InputChannel3
//     Standard Inputs/MAIN.IC02.T04/I @bit 3 <-> Module 1 (FSOES)/TxPDO/FSOE/InputChannel4
//     Standard Inputs/MAIN.IC02.T04/InfoData/State <-> InfoData/State
//   SODG11_SSCC610_2403701_PLC/SODG11_SSCC610_2403701_PLC Instance <-> EtherCAT Master (EtherCAT)/IC02.T01 (EK1100)/IC02.T05 (EL1904)
//     Standard Inputs/MAIN.IC02.T05/I <-> Module 1 (FSOES)/TxPDO/FSOE/InputChannel1
//     Standard Inputs/MAIN.IC02.T05/I @bit 1 <-> Module 1 (FSOES)/TxPDO/FSOE/InputChannel2
//     Standard Inputs/MAIN.IC02.T05/I @bit 2 <-> Module 1 (FSOES)/TxPDO/FSOE/InputChannel3
//     Standard Inputs/MAIN.IC02.T05/I @bit 3 <-> Module 1 (FSOES)/TxPDO/FSOE/InputChannel4
//     Standard Inputs/MAIN.IC02.T05/InfoData/State <-> InfoData/State
//   SODG11_SSCC610_2403701_PLC/SODG11_SSCC610_2403701_PLC Instance <-> EtherCAT Master (EtherCAT)/IC02.T01 (EK1100)/IC02.T06 (EL1904)
//     Standard Inputs/MAIN.IC02.T06/I <-> Module 1 (FSOES)/TxPDO/FSOE/InputChannel1
//     Standard Inputs/MAIN.IC02.T06/I @bit 1 <-> Module 1 (FSOES)/TxPDO/FSOE/InputChannel2
//     Standard Inputs/MAIN.IC02.T06/I @bit 2 <-> Module 1 (FSOES)/TxPDO/FSOE/InputChannel3
//     Standard Inputs/MAIN.IC02.T06/I @bit 3 <-> Module 1 (FSOES)/TxPDO/FSOE/InputChannel4
//     Standard Inputs/MAIN.IC02.T06/InfoData/State <-> InfoData/State
//   SODG11_SSCC610_2403701_PLC/SODG11_SSCC610_2403701_PLC Instance <-> EtherCAT Master (EtherCAT)/IC02.T01 (EK1100)/IC02.T07 (EL1904)
//     Standard Inputs/MAIN.IC02.T07/I <-> Module 1 (FSOES)/TxPDO/FSOE/InputChannel1
//     Standard Inputs/MAIN.IC02.T07/I @bit 1 <-> Module 1 (FSOES)/TxPDO/FSOE/InputChannel2
//     Standard Inputs/MAIN.IC02.T07/I @bit 2 <-> Module 1 (FSOES)/TxPDO/FSOE/InputChannel3
//     Standard Inputs/MAIN.IC02.T07/I @bit 3 <-> Module 1 (FSOES)/TxPDO/FSOE/InputChannel4
//     Standard Inputs/MAIN.IC02.T07/InfoData/State <-> InfoData/State
//   SODG11_SSCC610_2403701_PLC/SODG11_SSCC610_2403701_PLC Instance <-> EtherCAT Master (EtherCAT)/IC02.T01 (EK1100)/IC02.T08 (EL1904)
//     Standard Inputs/MAIN.IC02.T08/I <-> Module 1 (FSOES)/TxPDO/FSOE/InputChannel1
//     Standard Inputs/MAIN.IC02.T08/I @bit 1 <-> Module 1 (FSOES)/TxPDO/FSOE/InputChannel2
//     Standard Inputs/MAIN.IC02.T08/I @bit 2 <-> Module 1 (FSOES)/TxPDO/FSOE/InputChannel3
//     Standard Inputs/MAIN.IC02.T08/I @bit 3 <-> Module 1 (FSOES)/TxPDO/FSOE/InputChannel4
//     Standard Inputs/MAIN.IC02.T08/InfoData/State <-> InfoData/State
//   SODG11_SSCC610_2403701_PLC/SODG11_SSCC610_2403701_PLC Instance <-> EtherCAT Master (EtherCAT)/IC02.T01 (EK1100)/IC02.T09 (EL2904)
//     Standard Inputs/MAIN.IC02.T09/InfoData/State <-> InfoData/State
//   SODG11_SSCC610_2403701_PLC/SODG11_SSCC610_2403701_PLC Instance <-> EtherCAT Master (EtherCAT)/IC02.T01 (EK1100)/IC02.T10 (EL2904)
//     Standard Inputs/MAIN.IC02.T10/InfoData/State <-> InfoData/State
//   SODG11_SSCC610_2403701_PLC/SODG11_SSCC610_2403701_PLC Instance <-> EtherCAT Master (EtherCAT)/IC02.T01 (EK1100)/IC02.T11 (EL9410)
//     Standard Inputs/MAIN.IC02.T11/InfoData/State <-> InfoData/State
//     Standard Inputs/MAIN.IC02.T11/Up_UnderVoltage <-> Status Up/Undervoltage
//     Standard Inputs/MAIN.IC02.T11/Us_Undervoltage <-> Status Us/Undervoltage
//     Standard Inputs/MAIN.IC02.T11/WcState <-> WcState/WcState
//   SODG11_SSCC610_2403701_PLC/SODG11_SSCC610_2403701_PLC Instance <-> EtherCAT Master (EtherCAT)/IC02.T01 (EK1100)/IC02.T12 (EL1004)
//     Standard Inputs/MAIN.IC02.T12/I <-> Channel 1/Input
//     Standard Inputs/MAIN.IC02.T12/I @bit 1 <-> Channel 2/Input
//     Standard Inputs/MAIN.IC02.T12/I @bit 2 <-> Channel 3/Input
//     Standard Inputs/MAIN.IC02.T12/I @bit 3 <-> Channel 4/Input
//     Standard Inputs/MAIN.IC02.T12/InfoData/State <-> InfoData/State
//   SODG11_SSCC610_2403701_PLC/SODG11_SSCC610_2403701_PLC Instance <-> EtherCAT Master (EtherCAT)/IC02.T01 (EK1100)/IC02.T13 (EL1004)
//     Standard Inputs/MAIN.IC02.T13/I <-> Channel 1/Input
//     Standard Inputs/MAIN.IC02.T13/I @bit 1 <-> Channel 2/Input
//     Standard Inputs/MAIN.IC02.T13/I @bit 2 <-> Channel 3/Input
//     Standard Inputs/MAIN.IC02.T13/I @bit 3 <-> Channel 4/Input
//     Standard Inputs/MAIN.IC02.T13/InfoData/State <-> InfoData/State
//   SODG11_SSCC610_2403701_PLC/SODG11_SSCC610_2403701_PLC Instance <-> EtherCAT Master (EtherCAT)/IC02.T01 (EK1100)/IC02.T14 (EL2008)
//     Standard Inputs/MAIN.IC02.T14_STAT/InfoData/State <-> InfoData/State
//     Standard Outputs/MAIN.IC02.T14/Q <-> Channel 1/Output
//     Standard Outputs/MAIN.IC02.T14/Q @bit 1 <-> Channel 2/Output
//     Standard Outputs/MAIN.IC02.T14/Q @bit 2 <-> Channel 3/Output
//     Standard Outputs/MAIN.IC02.T14/Q @bit 3 <-> Channel 4/Output
//     Standard Outputs/MAIN.IC02.T14/Q @bit 4 <-> Channel 5/Output
//     Standard Outputs/MAIN.IC02.T14/Q @bit 5 <-> Channel 6/Output
//     Standard Outputs/MAIN.IC02.T14/Q @bit 6 <-> Channel 7/Output
//     Standard Outputs/MAIN.IC02.T14/Q @bit 7 <-> Channel 8/Output
//   SODG11_SSCC610_2403701_PLC/SODG11_SSCC610_2403701_PLC Instance <-> EtherCAT Master (EtherCAT)/IC02.T01 (EK1100)/IC02.T15 (EL2622)
//     Standard Inputs/MAIN.IC02.T15_STAT/InfoData/State <-> InfoData/State
//     Standard Outputs/MAIN.IC02.T15/Q0 <-> Channel 1/Output
//     Standard Outputs/MAIN.IC02.T15/Q1 <-> Channel 2/Output
//   SODG11_SSCC610_2403701_PLC/SODG11_SSCC610_2403701_PLC Instance <-> EtherCAT Master (EtherCAT)/IC02.T01 (EK1100)/IC02.T16 (EK1122)
//     Standard Inputs/MAIN.IC02.T16/InfoData/State <-> InfoData/State
//   SODG11_SSCC610_2403701_PLC/SODG11_SSCC610_2403701_PLC Instance <-> EtherCAT Master (EtherCAT)/IC02.T01 (EK1100)/IC02.T16 (EK1122)/Fix03.N01 (EP1008-0002)
//     Standard Inputs/Fix03.N01/I <-> Channel 1/Input
//     Standard Inputs/Fix03.N01/I @bit 1 <-> Channel 2/Input
//     Standard Inputs/Fix03.N01/I @bit 2 <-> Channel 3/Input
//     Standard Inputs/Fix03.N01/I @bit 3 <-> Channel 4/Input
//     Standard Inputs/Fix03.N01/I @bit 4 <-> Channel 5/Input
//     Standard Inputs/Fix03.N01/I @bit 5 <-> Channel 6/Input
//     Standard Inputs/Fix03.N01/I @bit 6 <-> Channel 7/Input
//     Standard Inputs/Fix03.N01/I @bit 7 <-> Channel 8/Input
//     Standard Inputs/Fix03.N01/InfoData/State <-> InfoData/State
//     Standard Inputs/Fix03.N01/Wc_State <-> WcState/WcState
//   SODG11_SSCC610_2403701_PLC/SODG11_SSCC610_2403701_PLC Instance <-> EtherCAT Master (EtherCAT)/IC02.T01 (EK1100)/IC02.T16 (EK1122)/Fix03.N02 (EP1008-0002)
//     Standard Inputs/Fix03.N02/I <-> Channel 1/Input
//     Standard Inputs/Fix03.N02/I @bit 1 <-> Channel 2/Input
//     Standard Inputs/Fix03.N02/I @bit 2 <-> Channel 3/Input
//     Standard Inputs/Fix03.N02/I @bit 3 <-> Channel 4/Input
//     Standard Inputs/Fix03.N02/I @bit 4 <-> Channel 5/Input
//     Standard Inputs/Fix03.N02/I @bit 5 <-> Channel 6/Input
//     Standard Inputs/Fix03.N02/I @bit 6 <-> Channel 7/Input
//     Standard Inputs/Fix03.N02/I @bit 7 <-> Channel 8/Input
//     Standard Inputs/Fix03.N02/InfoData/State <-> InfoData/State
//     Standard Inputs/Fix03.N02/Wc_State <-> WcState/WcState
//   SODG11_SSCC610_2403701_PLC/SODG11_SSCC610_2403701_PLC Instance <-> EtherCAT Master (EtherCAT)/IC02.T01 (EK1100)/IC02.T16 (EK1122)/Fix03.N03 (EP1008-0002)
//     Standard Inputs/Fix03.N03/I <-> Channel 1/Input
//     Standard Inputs/Fix03.N03/I @bit 1 <-> Channel 2/Input
//     Standard Inputs/Fix03.N03/I @bit 2 <-> Channel 3/Input
//     Standard Inputs/Fix03.N03/I @bit 3 <-> Channel 4/Input
//     Standard Inputs/Fix03.N03/I @bit 4 <-> Channel 5/Input
//     Standard Inputs/Fix03.N03/I @bit 5 <-> Channel 6/Input
//     Standard Inputs/Fix03.N03/I @bit 6 <-> Channel 7/Input
//     Standard Inputs/Fix03.N03/I @bit 7 <-> Channel 8/Input
//     Standard Inputs/Fix03.N03/InfoData/State <-> InfoData/State
//     Standard Inputs/Fix03.N03/Wc_State <-> WcState/WcState
//   SODG11_SSCC610_2403701_PLC/SODG11_SSCC610_2403701_PLC Instance <-> EtherCAT Master (EtherCAT)/IC02.T01 (EK1100)/IC02.T16 (EK1122)/Fix03.N04 (EP1008-0002)
//     Standard Inputs/Fix03.N04/I <-> Channel 1/Input
//     Standard Inputs/Fix03.N04/I @bit 1 <-> Channel 2/Input
//     Standard Inputs/Fix03.N04/I @bit 2 <-> Channel 3/Input
//     Standard Inputs/Fix03.N04/I @bit 3 <-> Channel 4/Input
//     Standard Inputs/Fix03.N04/I @bit 4 <-> Channel 5/Input
//     Standard Inputs/Fix03.N04/I @bit 5 <-> Channel 6/Input
//     Standard Inputs/Fix03.N04/I @bit 6 <-> Channel 7/Input
//     Standard Inputs/Fix03.N04/I @bit 7 <-> Channel 8/Input
//     Standard Inputs/Fix03.N04/InfoData/State <-> InfoData/State
//     Standard Inputs/Fix03.N04/Wc_State <-> WcState/WcState
//   SODG11_SSCC610_2403701_PLC/SODG11_SSCC610_2403701_PLC Instance <-> EtherCAT Master (EtherCAT)/IC02.T01 (EK1100)/IC02.T16 (EK1122)/Fix03.N05 (EP1008-0002)
//     Standard Inputs/Fix03.N05/I <-> Channel 1/Input
//     Standard Inputs/Fix03.N05/I @bit 1 <-> Channel 2/Input
//     Standard Inputs/Fix03.N05/I @bit 2 <-> Channel 3/Input
//     Standard Inputs/Fix03.N05/I @bit 3 <-> Channel 4/Input
//     Standard Inputs/Fix03.N05/I @bit 4 <-> Channel 5/Input
//     Standard Inputs/Fix03.N05/I @bit 5 <-> Channel 6/Input
//     Standard Inputs/Fix03.N05/I @bit 6 <-> Channel 7/Input
//     Standard Inputs/Fix03.N05/I @bit 7 <-> Channel 8/Input
//     Standard Inputs/Fix03.N05/InfoData/State <-> InfoData/State
//     Standard Inputs/Fix03.N05/Wc_State <-> WcState/WcState
//   SODG11_SSCC610_2403701_PLC/SODG11_SSCC610_2403701_PLC Instance <-> EtherCAT Master (EtherCAT)/IC02.T01 (EK1100)/IC02.T16 (EK1122)/Fix03.N06 (EP1008-0002)
//     Standard Inputs/Fix03.N06/I <-> Channel 1/Input
//     Standard Inputs/Fix03.N06/I @bit 1 <-> Channel 2/Input
//     Standard Inputs/Fix03.N06/I @bit 2 <-> Channel 3/Input
//     Standard Inputs/Fix03.N06/I @bit 3 <-> Channel 4/Input
//     Standard Inputs/Fix03.N06/I @bit 4 <-> Channel 5/Input
//     Standard Inputs/Fix03.N06/I @bit 5 <-> Channel 6/Input
//     Standard Inputs/Fix03.N06/I @bit 6 <-> Channel 7/Input
//     Standard Inputs/Fix03.N06/I @bit 7 <-> Channel 8/Input
//     Standard Inputs/Fix03.N06/InfoData/State <-> InfoData/State
//     Standard Inputs/Fix03.N06/Wc_State <-> WcState/WcState
//   SODG11_SSCC610_2403701_PLC/SODG11_SSCC610_2403701_PLC Instance <-> EtherCAT Master (EtherCAT)/IC02.T01 (EK1100)/IC02.T16 (EK1122)/Fix03.N07 (EP1008-0002)
//     Standard Inputs/Fix03.N07/I <-> Channel 1/Input
//     Standard Inputs/Fix03.N07/I @bit 1 <-> Channel 2/Input
//     Standard Inputs/Fix03.N07/I @bit 2 <-> Channel 3/Input
//     Standard Inputs/Fix03.N07/I @bit 3 <-> Channel 4/Input
//     Standard Inputs/Fix03.N07/I @bit 4 <-> Channel 5/Input
//     Standard Inputs/Fix03.N07/I @bit 5 <-> Channel 6/Input
//     Standard Inputs/Fix03.N07/I @bit 6 <-> Channel 7/Input
//     Standard Inputs/Fix03.N07/I @bit 7 <-> Channel 8/Input
//     Standard Inputs/Fix03.N07/InfoData/State <-> InfoData/State
//     Standard Inputs/Fix03.N07/Wc_State <-> WcState/WcState
//   SODG11_SSCC610_2403701_PLC/SODG11_SSCC610_2403701_PLC Instance <-> EtherCAT Master (EtherCAT)/IC02.T01 (EK1100)/IC02.T16 (EK1122)/Fix03.N08 (EP1008-0002)
//     Standard Inputs/Fix03.N08/I <-> Channel 1/Input
//     Standard Inputs/Fix03.N08/I @bit 1 <-> Channel 2/Input
//     Standard Inputs/Fix03.N08/I @bit 2 <-> Channel 3/Input
//     Standard Inputs/Fix03.N08/I @bit 3 <-> Channel 4/Input
//     Standard Inputs/Fix03.N08/I @bit 4 <-> Channel 5/Input
//     Standard Inputs/Fix03.N08/I @bit 5 <-> Channel 6/Input
//     Standard Inputs/Fix03.N08/I @bit 6 <-> Channel 7/Input
//     Standard Inputs/Fix03.N08/I @bit 7 <-> Channel 8/Input
//     Standard Inputs/Fix03.N08/InfoData/State <-> InfoData/State
//     Standard Inputs/Fix03.N08/Wc_State <-> WcState/WcState
//   SODG11_SSCC610_2403701_PLC/SODG11_SSCC610_2403701_PLC Instance <-> EtherCAT Master (EtherCAT)/IC02.T01 (EK1100)/IC02.T16 (EK1122)/Fix03.N09 (EP1008-0002)
//     Standard Inputs/Fix03.N09/I <-> Channel 1/Input
//     Standard Inputs/Fix03.N09/I @bit 1 <-> Channel 2/Input
//     Standard Inputs/Fix03.N09/I @bit 2 <-> Channel 3/Input
//     Standard Inputs/Fix03.N09/I @bit 3 <-> Channel 4/Input
//     Standard Inputs/Fix03.N09/I @bit 4 <-> Channel 5/Input
//     Standard Inputs/Fix03.N09/I @bit 5 <-> Channel 6/Input
//     Standard Inputs/Fix03.N09/I @bit 6 <-> Channel 7/Input
//     Standard Inputs/Fix03.N09/I @bit 7 <-> Channel 8/Input
//     Standard Inputs/Fix03.N09/InfoData/State <-> InfoData/State
//     Standard Inputs/Fix03.N09/Wc_State <-> WcState/WcState
//   SODG11_SSCC610_2403701_PLC/SODG11_SSCC610_2403701_PLC Instance <-> EtherCAT Master (EtherCAT)/IC02.T01 (EK1100)/IC02.T16 (EK1122)/Fix03.N10 (EP1008-0002)
//     Standard Inputs/Fix03.N10/I <-> Channel 1/Input
//     Standard Inputs/Fix03.N10/I @bit 1 <-> Channel 2/Input
//     Standard Inputs/Fix03.N10/I @bit 2 <-> Channel 3/Input
//     Standard Inputs/Fix03.N10/I @bit 3 <-> Channel 4/Input
//     Standard Inputs/Fix03.N10/I @bit 4 <-> Channel 5/Input
//     Standard Inputs/Fix03.N10/I @bit 5 <-> Channel 6/Input
//     Standard Inputs/Fix03.N10/I @bit 6 <-> Channel 7/Input
//     Standard Inputs/Fix03.N10/I @bit 7 <-> Channel 8/Input
//     Standard Inputs/Fix03.N10/InfoData/State <-> InfoData/State
//     Standard Inputs/Fix03.N10/Wc_State <-> WcState/WcState
//   SODG11_SSCC610_2403701_PLC/SODG11_SSCC610_2403701_PLC Instance <-> EtherCAT Master (EtherCAT)/IC02.T01 (EK1100)/IC02.T16 (EK1122)/Fix03.N100 (EX260-SEC1)
//     Standard Inputs/Fix03.N100_STAT/InfoData/State <-> InfoData/State
//     Standard Outputs/Fix03.N100/Q <-> Byte 0/Output
//     Standard Outputs/Fix03.N100/Q @bit 8 <-> Byte 1/Output
//     Standard Outputs/Fix03.N100/Q @bit 16 <-> Byte 2/Output
//     Standard Outputs/Fix03.N100/Q @bit 24 <-> Byte 3/Output
//   SODG11_SSCC610_2403701_PLC/SODG11_SSCC610_2403701_PLC Instance <-> EtherCAT Master (EtherCAT)/IC02.T01 (EK1100)/IC02.T16 (EK1122)/Fix03.N11 (EP1008-0002)
//     Standard Inputs/Fix03.N11/I <-> Channel 1/Input
//     Standard Inputs/Fix03.N11/I @bit 1 <-> Channel 2/Input
//     Standard Inputs/Fix03.N11/I @bit 2 <-> Channel 3/Input
//     Standard Inputs/Fix03.N11/I @bit 3 <-> Channel 4/Input
//     Standard Inputs/Fix03.N11/I @bit 4 <-> Channel 5/Input
//     Standard Inputs/Fix03.N11/I @bit 5 <-> Channel 6/Input
//     Standard Inputs/Fix03.N11/I @bit 6 <-> Channel 7/Input
//     Standard Inputs/Fix03.N11/I @bit 7 <-> Channel 8/Input
//     Standard Inputs/Fix03.N11/InfoData/State <-> InfoData/State
//     Standard Inputs/Fix03.N11/Wc_State <-> WcState/WcState
//   SODG11_SSCC610_2403701_PLC/SODG11_SSCC610_2403701_PLC Instance <-> EtherCAT Master (EtherCAT)/IC02.T01 (EK1100)/IC02.T16 (EK1122)/Fix03.N12 (EP1008-0002)
//     Standard Inputs/Fix03.N12/I <-> Channel 1/Input
//     Standard Inputs/Fix03.N12/I @bit 1 <-> Channel 2/Input
//     Standard Inputs/Fix03.N12/I @bit 2 <-> Channel 3/Input
//     Standard Inputs/Fix03.N12/I @bit 3 <-> Channel 4/Input
//     Standard Inputs/Fix03.N12/I @bit 4 <-> Channel 5/Input
//     Standard Inputs/Fix03.N12/I @bit 5 <-> Channel 6/Input
//     Standard Inputs/Fix03.N12/I @bit 6 <-> Channel 7/Input
//     Standard Inputs/Fix03.N12/I @bit 7 <-> Channel 8/Input
//     Standard Inputs/Fix03.N12/InfoData/State <-> InfoData/State
//     Standard Inputs/Fix03.N12/Wc_State <-> WcState/WcState
//   SODG11_SSCC610_2403701_PLC/SODG11_SSCC610_2403701_PLC Instance <-> EtherCAT Master (EtherCAT)/IC02.T01 (EK1100)/IC02.T16 (EK1122)/Fix03.N13 (EP1008-0002)
//     Standard Inputs/Fix03.N13/I <-> Channel 1/Input
//     Standard Inputs/Fix03.N13/I @bit 1 <-> Channel 2/Input
//     Standard Inputs/Fix03.N13/I @bit 2 <-> Channel 3/Input
//     Standard Inputs/Fix03.N13/I @bit 3 <-> Channel 4/Input
//     Standard Inputs/Fix03.N13/I @bit 4 <-> Channel 5/Input
//     Standard Inputs/Fix03.N13/I @bit 5 <-> Channel 6/Input
//     Standard Inputs/Fix03.N13/I @bit 6 <-> Channel 7/Input
//     Standard Inputs/Fix03.N13/I @bit 7 <-> Channel 8/Input
//     Standard Inputs/Fix03.N13/InfoData/State <-> InfoData/State
//     Standard Inputs/Fix03.N13/Wc_State <-> WcState/WcState
//   SODG11_SSCC610_2403701_PLC/SODG11_SSCC610_2403701_PLC Instance <-> EtherCAT Master (EtherCAT)/IC02.T01 (EK1100)/IC02.T16 (EK1122)/Fix03.N14 (EP1008-0002)
//     Standard Inputs/Fix03.N14/I <-> Channel 1/Input
//     Standard Inputs/Fix03.N14/I @bit 1 <-> Channel 2/Input
//     Standard Inputs/Fix03.N14/I @bit 2 <-> Channel 3/Input
//     Standard Inputs/Fix03.N14/I @bit 3 <-> Channel 4/Input
//     Standard Inputs/Fix03.N14/I @bit 4 <-> Channel 5/Input
//     Standard Inputs/Fix03.N14/I @bit 5 <-> Channel 6/Input
//     Standard Inputs/Fix03.N14/I @bit 6 <-> Channel 7/Input
//     Standard Inputs/Fix03.N14/I @bit 7 <-> Channel 8/Input
//     Standard Inputs/Fix03.N14/InfoData/State <-> InfoData/State
//     Standard Inputs/Fix03.N14/Wc_State <-> WcState/WcState
//   SODG11_SSCC610_2403701_PLC/SODG11_SSCC610_2403701_PLC Instance <-> EtherCAT Master (EtherCAT)/IC02.T01 (EK1100)/IC02.T16 (EK1122)/Fix03.N15 (EP1008-0002)
//     Standard Inputs/Fix03.N15/I <-> Channel 1/Input
//     Standard Inputs/Fix03.N15/I @bit 1 <-> Channel 2/Input
//     Standard Inputs/Fix03.N15/I @bit 2 <-> Channel 3/Input
//     Standard Inputs/Fix03.N15/I @bit 3 <-> Channel 4/Input
//     Standard Inputs/Fix03.N15/I @bit 4 <-> Channel 5/Input
//     Standard Inputs/Fix03.N15/I @bit 5 <-> Channel 6/Input
//     Standard Inputs/Fix03.N15/I @bit 6 <-> Channel 7/Input
//     Standard Inputs/Fix03.N15/I @bit 7 <-> Channel 8/Input
//     Standard Inputs/Fix03.N15/InfoData/State <-> InfoData/State
//     Standard Inputs/Fix03.N15/Wc_State <-> WcState/WcState
//   SODG11_SSCC610_2403701_PLC/SODG11_SSCC610_2403701_PLC Instance <-> EtherCAT Master (EtherCAT)/IC02.T01 (EK1100)/IC02.T16 (EK1122)/Fix03.N16 (EP1008-0002)
//     Standard Inputs/Fix03.N16/I <-> Channel 1/Input
//     Standard Inputs/Fix03.N16/I @bit 1 <-> Channel 2/Input
//     Standard Inputs/Fix03.N16/I @bit 2 <-> Channel 3/Input
//     Standard Inputs/Fix03.N16/I @bit 3 <-> Channel 4/Input
//     Standard Inputs/Fix03.N16/I @bit 4 <-> Channel 5/Input
//     Standard Inputs/Fix03.N16/I @bit 5 <-> Channel 6/Input
//     Standard Inputs/Fix03.N16/I @bit 6 <-> Channel 7/Input
//     Standard Inputs/Fix03.N16/I @bit 7 <-> Channel 8/Input
//     Standard Inputs/Fix03.N16/InfoData/State <-> InfoData/State
//     Standard Inputs/Fix03.N16/Wc_State <-> WcState/WcState
//   SODG11_SSCC610_2403701_PLC/SODG11_SSCC610_2403701_PLC Instance <-> EtherCAT Master (EtherCAT)/IC02.T01 (EK1100)/IC02.T16 (EK1122)/Fix03.N17 (EP1008-0002)
//     Standard Inputs/Fix03.N17/I <-> Channel 1/Input
//     Standard Inputs/Fix03.N17/I @bit 1 <-> Channel 2/Input
//     Standard Inputs/Fix03.N17/I @bit 2 <-> Channel 3/Input
//     Standard Inputs/Fix03.N17/I @bit 3 <-> Channel 4/Input
//     Standard Inputs/Fix03.N17/I @bit 4 <-> Channel 5/Input
//     Standard Inputs/Fix03.N17/I @bit 5 <-> Channel 6/Input
//     Standard Inputs/Fix03.N17/I @bit 6 <-> Channel 7/Input
//     Standard Inputs/Fix03.N17/I @bit 7 <-> Channel 8/Input
//     Standard Inputs/Fix03.N17/InfoData/State <-> InfoData/State
//     Standard Inputs/Fix03.N17/Wc_State <-> WcState/WcState
//   SODG11_SSCC610_2403701_PLC/SODG11_SSCC610_2403701_PLC Instance <-> EtherCAT Master (EtherCAT)/IC02.T01 (EK1100)/IC02.T16 (EK1122)/Fix03.N18 (EP1008-0002)
//     Standard Inputs/Fix03.N18/I <-> Channel 1/Input
//     Standard Inputs/Fix03.N18/I @bit 1 <-> Channel 2/Input
//     Standard Inputs/Fix03.N18/I @bit 2 <-> Channel 3/Input
//     Standard Inputs/Fix03.N18/I @bit 3 <-> Channel 4/Input
//     Standard Inputs/Fix03.N18/I @bit 4 <-> Channel 5/Input
//     Standard Inputs/Fix03.N18/I @bit 5 <-> Channel 6/Input
//     Standard Inputs/Fix03.N18/I @bit 6 <-> Channel 7/Input
//     Standard Inputs/Fix03.N18/I @bit 7 <-> Channel 8/Input
//     Standard Inputs/Fix03.N18/InfoData/State <-> InfoData/State
//     Standard Inputs/Fix03.N18/Wc_State <-> WcState/WcState
//   SODG11_SSCC610_2403701_PLC/SODG11_SSCC610_2403701_PLC Instance <-> EtherCAT Master (EtherCAT)/IC02.T01 (EK1100)/IC02.T16 (EK1122)/Fix03.N19 (EP1008-0002)
//     Standard Inputs/Fix03.N19/I <-> Channel 1/Input
//     Standard Inputs/Fix03.N19/I @bit 1 <-> Channel 2/Input
//     Standard Inputs/Fix03.N19/I @bit 2 <-> Channel 3/Input
//     Standard Inputs/Fix03.N19/I @bit 3 <-> Channel 4/Input
//     Standard Inputs/Fix03.N19/I @bit 4 <-> Channel 5/Input
//     Standard Inputs/Fix03.N19/I @bit 5 <-> Channel 6/Input
//     Standard Inputs/Fix03.N19/I @bit 6 <-> Channel 7/Input
//     Standard Inputs/Fix03.N19/I @bit 7 <-> Channel 8/Input
//     Standard Inputs/Fix03.N19/InfoData/State <-> InfoData/State
//     Standard Inputs/Fix03.N19/Wc_State <-> WcState/WcState
//   SODG11_SSCC610_2403701_PLC/SODG11_SSCC610_2403701_PLC Instance <-> EtherCAT Master (EtherCAT)/IC02.T01 (EK1100)/IC02.T16 (EK1122)/Fix03.N20 (EP1008-0002)
//     Standard Inputs/Fix03.N20/I <-> Channel 1/Input
//     Standard Inputs/Fix03.N20/I @bit 1 <-> Channel 2/Input
//     Standard Inputs/Fix03.N20/I @bit 2 <-> Channel 3/Input
//     Standard Inputs/Fix03.N20/I @bit 3 <-> Channel 4/Input
//     Standard Inputs/Fix03.N20/I @bit 4 <-> Channel 5/Input
//     Standard Inputs/Fix03.N20/I @bit 5 <-> Channel 6/Input
//     Standard Inputs/Fix03.N20/I @bit 6 <-> Channel 7/Input
//     Standard Inputs/Fix03.N20/I @bit 7 <-> Channel 8/Input
//     Standard Inputs/Fix03.N20/InfoData/State <-> InfoData/State
//     Standard Inputs/Fix03.N20/Wc_State <-> WcState/WcState
//   SODG11_SSCC610_2403701_PLC/SODG11_SSCC610_2403701_PLC Instance <-> EtherCAT Master (EtherCAT)/IC02.T01 (EK1100)/IC02.T16 (EK1122)/Fix03.N21 (EP1008-0002)
//     Standard Inputs/Fix03.N21/I <-> Channel 1/Input
//     Standard Inputs/Fix03.N21/I @bit 1 <-> Channel 2/Input
//     Standard Inputs/Fix03.N21/I @bit 2 <-> Channel 3/Input
//     Standard Inputs/Fix03.N21/I @bit 3 <-> Channel 4/Input
//     Standard Inputs/Fix03.N21/I @bit 4 <-> Channel 5/Input
//     Standard Inputs/Fix03.N21/I @bit 5 <-> Channel 6/Input
//     Standard Inputs/Fix03.N21/I @bit 6 <-> Channel 7/Input
//     Standard Inputs/Fix03.N21/I @bit 7 <-> Channel 8/Input
//     Standard Inputs/Fix03.N21/InfoData/State <-> InfoData/State
//     Standard Inputs/Fix03.N21/Wc_State <-> WcState/WcState
//   SODG11_SSCC610_2403701_PLC/SODG11_SSCC610_2403701_PLC Instance <-> EtherCAT Master (EtherCAT)/IC02.T01 (EK1100)/IC02.T16 (EK1122)/Fix03.N22 (EP1008-0002)
//     Standard Inputs/Fix03.N22/I <-> Channel 1/Input
//     Standard Inputs/Fix03.N22/I @bit 1 <-> Channel 2/Input
//     Standard Inputs/Fix03.N22/I @bit 2 <-> Channel 3/Input
//     Standard Inputs/Fix03.N22/I @bit 3 <-> Channel 4/Input
//     Standard Inputs/Fix03.N22/I @bit 4 <-> Channel 5/Input
//     Standard Inputs/Fix03.N22/I @bit 5 <-> Channel 6/Input
//     Standard Inputs/Fix03.N22/I @bit 6 <-> Channel 7/Input
//     Standard Inputs/Fix03.N22/I @bit 7 <-> Channel 8/Input
//     Standard Inputs/Fix03.N22/InfoData/State <-> InfoData/State
//     Standard Inputs/Fix03.N22/Wc_State <-> WcState/WcState
//   SODG11_SSCC610_2403701_PLC/SODG11_SSCC610_2403701_PLC Instance <-> EtherCAT Master (EtherCAT)/IC02.T01 (EK1100)/IC02.T16 (EK1122)/Fix03.N90 (EP9214-0023)
//     Standard Inputs/Fix03.N90_STAT/Channel_1/Channel_Error <-> DPO Inputs Channel 1/Channel Error
//     Standard Inputs/Fix03.N90_STAT/Channel_2/Channel_Error <-> DPO Inputs Channel 2/Channel Error
//     Standard Inputs/Fix03.N90_STAT/Channel_3/Channel_Error <-> DPO Inputs Channel 3/Channel Error
//     Standard Inputs/Fix03.N90_STAT/Channel_4/Channel_Error <-> DPO Inputs Channel 4/Channel Error
//     Standard Inputs/Fix03.N90_STAT/Channel_1/Error_Up <-> DPO Inputs Channel 1/Error Up
//     Standard Inputs/Fix03.N90_STAT/Channel_2/Error_Up <-> DPO Inputs Channel 2/Error Up
//     Standard Inputs/Fix03.N90_STAT/Channel_3/Error_Up <-> DPO Inputs Channel 3/Error Up
//     Standard Inputs/Fix03.N90_STAT/Channel_4/Error_Up <-> DPO Inputs Channel 4/Error Up
//     Standard Inputs/Fix03.N90_STAT/Channel_1/Error_Us <-> DPO Inputs Channel 1/Error Us
//     Standard Inputs/Fix03.N90_STAT/Channel_2/Error_Us <-> DPO Inputs Channel 2/Error Us
//     Standard Inputs/Fix03.N90_STAT/Channel_3/Error_Us <-> DPO Inputs Channel 3/Error Us
//     Standard Inputs/Fix03.N90_STAT/Channel_4/Error_Us <-> DPO Inputs Channel 4/Error Us
//     Standard Inputs/Fix03.N90_STAT/Channel_1/Status_Up <-> DPO Inputs Channel 1/Status Up
//     Standard Inputs/Fix03.N90_STAT/Channel_2/Status_Up <-> DPO Inputs Channel 2/Status Up
//     Standard Inputs/Fix03.N90_STAT/Channel_3/Status_Up <-> DPO Inputs Channel 3/Status Up
//     Standard Inputs/Fix03.N90_STAT/Channel_4/Status_Up <-> DPO Inputs Channel 4/Status Up
//     Standard Inputs/Fix03.N90_STAT/Channel_1/Status_Us <-> DPO Inputs Channel 1/Status Us
//     Standard Inputs/Fix03.N90_STAT/Channel_2/Status_Us <-> DPO Inputs Channel 2/Status Us
//     Standard Inputs/Fix03.N90_STAT/Channel_3/Status_Us <-> DPO Inputs Channel 3/Status Us
//     Standard Inputs/Fix03.N90_STAT/Channel_4/Status_Us <-> DPO Inputs Channel 4/Status Us
//     Standard Inputs/Fix03.N90_STAT/Channel_1/SyncError <-> DPO Inputs Channel 1/Sync error
//     Standard Inputs/Fix03.N90_STAT/Channel_2/SyncError <-> DPO Inputs Channel 2/Sync error
//     Standard Inputs/Fix03.N90_STAT/Channel_3/SyncError <-> DPO Inputs Channel 3/Sync error
//     Standard Inputs/Fix03.N90_STAT/Channel_4/SyncError <-> DPO Inputs Channel 4/Sync error
//     Standard Inputs/Fix03.N90_STAT/Channel_1/TxPDO_State <-> DPO Inputs Channel 1/TxPDO State
//     Standard Inputs/Fix03.N90_STAT/Channel_2/TxPDO_State <-> DPO Inputs Channel 2/TxPDO State
//     Standard Inputs/Fix03.N90_STAT/Channel_3/TxPDO_State <-> DPO Inputs Channel 3/TxPDO State
//     Standard Inputs/Fix03.N90_STAT/Channel_4/TxPDO_State <-> DPO Inputs Channel 4/TxPDO State
//     Standard Inputs/Fix03.N90_STAT/Channel_1/TxPDO_Toggle <-> DPO Inputs Channel 1/TxPDO Toggle
//     Standard Inputs/Fix03.N90_STAT/Channel_2/TxPDO_Toggle <-> DPO Inputs Channel 2/TxPDO Toggle
//     Standard Inputs/Fix03.N90_STAT/Channel_3/TxPDO_Toggle <-> DPO Inputs Channel 3/TxPDO Toggle
//     Standard Inputs/Fix03.N90_STAT/Channel_4/TxPDO_Toggle <-> DPO Inputs Channel 4/TxPDO Toggle
//     Standard Inputs/Fix03.N90_STAT/Channel_1/Warning_Up <-> DPO Inputs Channel 1/Warning Up
//     Standard Inputs/Fix03.N90_STAT/Channel_2/Warning_Up <-> DPO Inputs Channel 2/Warning Up
//     Standard Inputs/Fix03.N90_STAT/Channel_3/Warning_Up <-> DPO Inputs Channel 3/Warning Up
//     Standard Inputs/Fix03.N90_STAT/Channel_4/Warning_Up <-> DPO Inputs Channel 4/Warning Up
//     Standard Inputs/Fix03.N90_STAT/Channel_1/Warning_Us <-> DPO Inputs Channel 1/Warning Us
//     Standard Inputs/Fix03.N90_STAT/Channel_2/Warning_Us <-> DPO Inputs Channel 2/Warning Us
//     Standard Inputs/Fix03.N90_STAT/Channel_3/Warning_Us <-> DPO Inputs Channel 3/Warning Us
//     Standard Inputs/Fix03.N90_STAT/Channel_4/Warning_Us <-> DPO Inputs Channel 4/Warning Us
//     Standard Inputs/Fix03.N90_STAT/Device/Global_Error_Bit <-> DPO Inputs Device/Global Error Bit
//     Standard Inputs/Fix03.N90_STAT/Device/Reset_Input <-> DPO Inputs Device/Reset Input
//     Standard Inputs/Fix03.N90_STAT/Device/Temperature_Error <-> DPO Inputs Device/Temperature Error
//     Standard Inputs/Fix03.N90_STAT/Device/Temperature_Warning <-> DPO Inputs Device/Temperature Warning
//     Standard Inputs/Fix03.N90_STAT/Device/TxPDO_State <-> DPO Inputs Device/TxPDO State
//     Standard Inputs/Fix03.N90_STAT/Device/TxPDO_Toggle <-> DPO Inputs Device/TxPDO Toggle
//     Standard Inputs/Fix03.N90_STAT/Device/Up_Error <-> DPO Inputs Device/Up Error
//     Standard Inputs/Fix03.N90_STAT/Device/Up_Warning <-> DPO Inputs Device/Up Warning
//     Standard Inputs/Fix03.N90_STAT/Device/Us_Error <-> DPO Inputs Device/Us Error
//     Standard Inputs/Fix03.N90_STAT/Device/Us_Warning <-> DPO Inputs Device/Us Warning
//     Standard Inputs/Fix03.N90_STAT/InfoData/AdsAddr <-> InfoData/AdsAddr
//     Standard Inputs/Fix03.N90_STAT/InfoData/State <-> InfoData/State
//     Standard Inputs/Fix03.N90_STAT/Wc_State <-> WcState/WcState
//     Standard Outputs/Fix03.N90_CMD/Channel1/Output_Up <-> DPO Outputs Channel 1/Output Up
//     Standard Outputs/Fix03.N90_CMD/Channel2/Output_Up <-> DPO Outputs Channel 2/Output Up
//     Standard Outputs/Fix03.N90_CMD/Channel2/Output_Up <-> DPO Outputs Channel 3/Output Up
//     Standard Outputs/Fix03.N90_CMD/Channel4/Output_Up <-> DPO Outputs Channel 4/Output Up
//     Standard Outputs/Fix03.N90_CMD/Channel1/Output_Us <-> DPO Outputs Channel 1/Output Us
//     Standard Outputs/Fix03.N90_CMD/Channel2/Output_Us <-> DPO Outputs Channel 2/Output Us
//     Standard Outputs/Fix03.N90_CMD/Channel3/Output_Us <-> DPO Outputs Channel 3/Output Us
//     Standard Outputs/Fix03.N90_CMD/Channel4/Output_Us <-> DPO Outputs Channel 4/Output Us
//     Standard Outputs/Fix03.N90_CMD/Channel1/Reset_Up <-> DPO Outputs Channel 1/Reset Up
//     Standard Outputs/Fix03.N90_CMD/Channel2/Reset_Up <-> DPO Outputs Channel 2/Reset Up
//     Standard Outputs/Fix03.N90_CMD/Channel3/Reset_Up <-> DPO Outputs Channel 3/Reset Up
//     Standard Outputs/Fix03.N90_CMD/Channel4/Reset_Up <-> DPO Outputs Channel 4/Reset Up
//     Standard Outputs/Fix03.N90_CMD/Channel1/Reset_Us <-> DPO Outputs Channel 1/Reset Us
//     Standard Outputs/Fix03.N90_CMD/Channel2/Reset_Us <-> DPO Outputs Channel 2/Reset Us
//     Standard Outputs/Fix03.N90_CMD/Channel3/Reset_Us <-> DPO Outputs Channel 3/Reset Us
//     Standard Outputs/Fix03.N90_CMD/Channel4/Reset_Us <-> DPO Outputs Channel 4/Reset Us
//     Standard Outputs/Fix03.N90_CMD/Device/Enable_Control_Via_Fieldbus <-> DPO Outputs Device/Enable Control Via Fieldbus
//     Standard Outputs/Fix03.N90_CMD/Device/Global_Reset <-> DPO Outputs Device/Global Reset
//   SODG11_SSCC610_2403701_PLC/SODG11_SSCC610_2403701_PLC Instance <-> EtherCAT Master (EtherCAT)/IC02.T01 (EK1100)/IC02.T16 (EK1122)/Fix03.N98  (EP2328-0002)
//     Standard Inputs/Fix03.N98.I <-> Channel 1/Input
//     Standard Inputs/Fix03.N98.I @bit 1 <-> Channel 2/Input
//     Standard Inputs/Fix03.N98.I @bit 2 <-> Channel 3/Input
//     Standard Inputs/Fix03.N98.I @bit 3 <-> Channel 4/Input
//     Standard Inputs/Fix03.N98.State <-> InfoData/State
//     Standard Inputs/Fix03.N98.WC_State <-> WcState/WcState
//     Standard Outputs/Fix03.N98.Q <-> Channel 5/Output
//     Standard Outputs/Fix03.N98.Q @bit 1 <-> Channel 6/Output
//     Standard Outputs/Fix03.N98.Q @bit 2 <-> Channel 7/Output
//     Standard Outputs/Fix03.N98.Q @bit 3 <-> Channel 8/Output
//   SODG11_SSCC610_2403701_PLC/SODG11_SSCC610_2403701_PLC Instance <-> EtherCAT Master (EtherCAT)/IC02.T01 (EK1100)/IC02.T16 (EK1122)/Fix04.N01 (EP1008-0002)
//     Standard Inputs/Fix04.N01/I <-> Channel 1/Input
//     Standard Inputs/Fix04.N01/I @bit 1 <-> Channel 2/Input
//     Standard Inputs/Fix04.N01/I @bit 2 <-> Channel 3/Input
//     Standard Inputs/Fix04.N01/I @bit 3 <-> Channel 4/Input
//     Standard Inputs/Fix04.N01/I @bit 4 <-> Channel 5/Input
//     Standard Inputs/Fix04.N01/I @bit 5 <-> Channel 6/Input
//     Standard Inputs/Fix04.N01/I @bit 6 <-> Channel 7/Input
//     Standard Inputs/Fix04.N01/I @bit 7 <-> Channel 8/Input
//     Standard Inputs/Fix04.N01/InfoData/State <-> InfoData/State
//     Standard Inputs/Fix04.N01/Wc_State <-> WcState/WcState
//   SODG11_SSCC610_2403701_PLC/SODG11_SSCC610_2403701_PLC Instance <-> EtherCAT Master (EtherCAT)/IC02.T01 (EK1100)/IC02.T16 (EK1122)/Fix04.N02 (EP1008-0002)
//     Standard Inputs/Fix04.N02/I <-> Channel 1/Input
//     Standard Inputs/Fix04.N02/I @bit 1 <-> Channel 2/Input
//     Standard Inputs/Fix04.N02/I @bit 2 <-> Channel 3/Input
//     Standard Inputs/Fix04.N02/I @bit 3 <-> Channel 4/Input
//     Standard Inputs/Fix04.N02/I @bit 4 <-> Channel 5/Input
//     Standard Inputs/Fix04.N02/I @bit 5 <-> Channel 6/Input
//     Standard Inputs/Fix04.N02/I @bit 6 <-> Channel 7/Input
//     Standard Inputs/Fix04.N02/I @bit 7 <-> Channel 8/Input
//     Standard Inputs/Fix04.N02/InfoData/State <-> InfoData/State
//     Standard Inputs/Fix04.N02/Wc_State <-> WcState/WcState
//   SODG11_SSCC610_2403701_PLC/SODG11_SSCC610_2403701_PLC Instance <-> EtherCAT Master (EtherCAT)/IC02.T01 (EK1100)/IC02.T16 (EK1122)/Fix04.N03 (EP1008-0002)
//     Standard Inputs/Fix04.N03/I <-> Channel 1/Input
//     Standard Inputs/Fix04.N03/I @bit 1 <-> Channel 2/Input
//     Standard Inputs/Fix04.N03/I @bit 2 <-> Channel 3/Input
//     Standard Inputs/Fix04.N03/I @bit 3 <-> Channel 4/Input
//     Standard Inputs/Fix04.N03/I @bit 4 <-> Channel 5/Input
//     Standard Inputs/Fix04.N03/I @bit 5 <-> Channel 6/Input
//     Standard Inputs/Fix04.N03/I @bit 6 <-> Channel 7/Input
//     Standard Inputs/Fix04.N03/I @bit 7 <-> Channel 8/Input
//     Standard Inputs/Fix04.N03/InfoData/State <-> InfoData/State
//     Standard Inputs/Fix04.N03/Wc_State <-> WcState/WcState
//   SODG11_SSCC610_2403701_PLC/SODG11_SSCC610_2403701_PLC Instance <-> EtherCAT Master (EtherCAT)/IC02.T01 (EK1100)/IC02.T16 (EK1122)/Fix04.N04 (EP1008-0002)
//     Standard Inputs/Fix04.N04/I <-> Channel 1/Input
//     Standard Inputs/Fix04.N04/I @bit 1 <-> Channel 2/Input
//     Standard Inputs/Fix04.N04/I @bit 2 <-> Channel 3/Input
//     Standard Inputs/Fix04.N04/I @bit 3 <-> Channel 4/Input
//     Standard Inputs/Fix04.N04/I @bit 4 <-> Channel 5/Input
//     Standard Inputs/Fix04.N04/I @bit 5 <-> Channel 6/Input
//     Standard Inputs/Fix04.N04/I @bit 6 <-> Channel 7/Input
//     Standard Inputs/Fix04.N04/I @bit 7 <-> Channel 8/Input
//     Standard Inputs/Fix04.N04/InfoData/State <-> InfoData/State
//     Standard Inputs/Fix04.N04/Wc_State <-> WcState/WcState
//   SODG11_SSCC610_2403701_PLC/SODG11_SSCC610_2403701_PLC Instance <-> EtherCAT Master (EtherCAT)/IC02.T01 (EK1100)/IC02.T16 (EK1122)/Fix04.N05 (EP1008-0002)
//     Standard Inputs/Fix04.N05/I <-> Channel 1/Input
//     Standard Inputs/Fix04.N05/I @bit 1 <-> Channel 2/Input
//     Standard Inputs/Fix04.N05/I @bit 2 <-> Channel 3/Input
//     Standard Inputs/Fix04.N05/I @bit 3 <-> Channel 4/Input
//     Standard Inputs/Fix04.N05/I @bit 4 <-> Channel 5/Input
//     Standard Inputs/Fix04.N05/I @bit 5 <-> Channel 6/Input
//     Standard Inputs/Fix04.N05/I @bit 6 <-> Channel 7/Input
//     Standard Inputs/Fix04.N05/I @bit 7 <-> Channel 8/Input
//     Standard Inputs/Fix04.N05/InfoData/State <-> InfoData/State
//     Standard Inputs/Fix04.N05/Wc_State <-> WcState/WcState
//   SODG11_SSCC610_2403701_PLC/SODG11_SSCC610_2403701_PLC Instance <-> EtherCAT Master (EtherCAT)/IC02.T01 (EK1100)/IC02.T16 (EK1122)/Fix04.N06 (EP1008-0002)
//     Standard Inputs/Fix04.N06/I <-> Channel 1/Input
//     Standard Inputs/Fix04.N06/I @bit 1 <-> Channel 2/Input
//     Standard Inputs/Fix04.N06/I @bit 2 <-> Channel 3/Input
//     Standard Inputs/Fix04.N06/I @bit 3 <-> Channel 4/Input
//     Standard Inputs/Fix04.N06/I @bit 4 <-> Channel 5/Input
//     Standard Inputs/Fix04.N06/I @bit 5 <-> Channel 6/Input
//     Standard Inputs/Fix04.N06/I @bit 6 <-> Channel 7/Input
//     Standard Inputs/Fix04.N06/I @bit 7 <-> Channel 8/Input
//     Standard Inputs/Fix04.N06/InfoData/State <-> InfoData/State
//     Standard Inputs/Fix04.N06/Wc_State <-> WcState/WcState
//   SODG11_SSCC610_2403701_PLC/SODG11_SSCC610_2403701_PLC Instance <-> EtherCAT Master (EtherCAT)/IC02.T01 (EK1100)/IC02.T16 (EK1122)/Fix04.N07 (EP1008-0002)
//     Standard Inputs/Fix04.N07/I <-> Channel 1/Input
//     Standard Inputs/Fix04.N07/I @bit 1 <-> Channel 2/Input
//     Standard Inputs/Fix04.N07/I @bit 2 <-> Channel 3/Input
//     Standard Inputs/Fix04.N07/I @bit 3 <-> Channel 4/Input
//     Standard Inputs/Fix04.N07/I @bit 4 <-> Channel 5/Input
//     Standard Inputs/Fix04.N07/I @bit 5 <-> Channel 6/Input
//     Standard Inputs/Fix04.N07/I @bit 6 <-> Channel 7/Input
//     Standard Inputs/Fix04.N07/I @bit 7 <-> Channel 8/Input
//     Standard Inputs/Fix04.N07/InfoData/State <-> InfoData/State
//     Standard Inputs/Fix04.N07/Wc_State <-> WcState/WcState
//   SODG11_SSCC610_2403701_PLC/SODG11_SSCC610_2403701_PLC Instance <-> EtherCAT Master (EtherCAT)/IC02.T01 (EK1100)/IC02.T16 (EK1122)/Fix04.N08 (EP1008-0002)
//     Standard Inputs/Fix04.N08/I <-> Channel 1/Input
//     Standard Inputs/Fix04.N08/I @bit 1 <-> Channel 2/Input
//     Standard Inputs/Fix04.N08/I @bit 2 <-> Channel 3/Input
//     Standard Inputs/Fix04.N08/I @bit 3 <-> Channel 4/Input
//     Standard Inputs/Fix04.N08/I @bit 4 <-> Channel 5/Input
//     Standard Inputs/Fix04.N08/I @bit 5 <-> Channel 6/Input
//     Standard Inputs/Fix04.N08/I @bit 6 <-> Channel 7/Input
//     Standard Inputs/Fix04.N08/I @bit 7 <-> Channel 8/Input
//     Standard Inputs/Fix04.N08/InfoData/State <-> InfoData/State
//     Standard Inputs/Fix04.N08/Wc_State <-> WcState/WcState
//   SODG11_SSCC610_2403701_PLC/SODG11_SSCC610_2403701_PLC Instance <-> EtherCAT Master (EtherCAT)/IC02.T01 (EK1100)/IC02.T16 (EK1122)/Fix04.N09 (EP1008-0002)
//     Standard Inputs/Fix04.N09/I <-> Channel 1/Input
//     Standard Inputs/Fix04.N09/I @bit 1 <-> Channel 2/Input
//     Standard Inputs/Fix04.N09/I @bit 2 <-> Channel 3/Input
//     Standard Inputs/Fix04.N09/I @bit 3 <-> Channel 4/Input
//     Standard Inputs/Fix04.N09/I @bit 4 <-> Channel 5/Input
//     Standard Inputs/Fix04.N09/I @bit 5 <-> Channel 6/Input
//     Standard Inputs/Fix04.N09/I @bit 6 <-> Channel 7/Input
//     Standard Inputs/Fix04.N09/I @bit 7 <-> Channel 8/Input
//     Standard Inputs/Fix04.N09/InfoData/State <-> InfoData/State
//     Standard Inputs/Fix04.N09/Wc_State <-> WcState/WcState
//   SODG11_SSCC610_2403701_PLC/SODG11_SSCC610_2403701_PLC Instance <-> EtherCAT Master (EtherCAT)/IC02.T01 (EK1100)/IC02.T16 (EK1122)/Fix04.N10 (EP1008-0002)
//     Standard Inputs/Fix04.N10/I <-> Channel 1/Input
//     Standard Inputs/Fix04.N10/I @bit 1 <-> Channel 2/Input
//     Standard Inputs/Fix04.N10/I @bit 2 <-> Channel 3/Input
//     Standard Inputs/Fix04.N10/I @bit 3 <-> Channel 4/Input
//     Standard Inputs/Fix04.N10/I @bit 4 <-> Channel 5/Input
//     Standard Inputs/Fix04.N10/I @bit 5 <-> Channel 6/Input
//     Standard Inputs/Fix04.N10/I @bit 6 <-> Channel 7/Input
//     Standard Inputs/Fix04.N10/I @bit 7 <-> Channel 8/Input
//     Standard Inputs/Fix04.N10/InfoData/State <-> InfoData/State
//     Standard Inputs/Fix04.N10/Wc_State <-> WcState/WcState
//   SODG11_SSCC610_2403701_PLC/SODG11_SSCC610_2403701_PLC Instance <-> EtherCAT Master (EtherCAT)/IC02.T01 (EK1100)/IC02.T16 (EK1122)/Fix04.N100 (EX260-SEC1)
//     Standard Inputs/Fix04.N100_STAT/InfoData/State <-> InfoData/State
//     Standard Outputs/Fix04.N100/Q <-> Byte 0/Output
//     Standard Outputs/Fix04.N100/Q @bit 8 <-> Byte 1/Output
//     Standard Outputs/Fix04.N100/Q @bit 16 <-> Byte 2/Output
//     Standard Outputs/Fix04.N100/Q @bit 24 <-> Byte 3/Output
//   SODG11_SSCC610_2403701_PLC/SODG11_SSCC610_2403701_PLC Instance <-> EtherCAT Master (EtherCAT)/IC02.T01 (EK1100)/IC02.T16 (EK1122)/Fix04.N11 (EP1008-0002)
//     Standard Inputs/Fix04.N11/I <-> Channel 1/Input
//     Standard Inputs/Fix04.N11/I @bit 1 <-> Channel 2/Input
//     Standard Inputs/Fix04.N11/I @bit 2 <-> Channel 3/Input
//     Standard Inputs/Fix04.N11/I @bit 3 <-> Channel 4/Input
//     Standard Inputs/Fix04.N11/I @bit 4 <-> Channel 5/Input
//     Standard Inputs/Fix04.N11/I @bit 5 <-> Channel 6/Input
//     Standard Inputs/Fix04.N11/I @bit 6 <-> Channel 7/Input
//     Standard Inputs/Fix04.N11/I @bit 7 <-> Channel 8/Input
//     Standard Inputs/Fix04.N11/InfoData/State <-> InfoData/State
//     Standard Inputs/Fix04.N11/Wc_State <-> WcState/WcState
//   SODG11_SSCC610_2403701_PLC/SODG11_SSCC610_2403701_PLC Instance <-> EtherCAT Master (EtherCAT)/IC02.T01 (EK1100)/IC02.T16 (EK1122)/Fix04.N12 (EP1008-0002)
//     Standard Inputs/Fix04.N12/I <-> Channel 1/Input
//     Standard Inputs/Fix04.N12/I @bit 1 <-> Channel 2/Input
//     Standard Inputs/Fix04.N12/I @bit 2 <-> Channel 3/Input
//     Standard Inputs/Fix04.N12/I @bit 3 <-> Channel 4/Input
//     Standard Inputs/Fix04.N12/I @bit 4 <-> Channel 5/Input
//     Standard Inputs/Fix04.N12/I @bit 5 <-> Channel 6/Input
//     Standard Inputs/Fix04.N12/I @bit 6 <-> Channel 7/Input
//     Standard Inputs/Fix04.N12/I @bit 7 <-> Channel 8/Input
//     Standard Inputs/Fix04.N12/InfoData/State <-> InfoData/State
//     Standard Inputs/Fix04.N12/Wc_State <-> WcState/WcState
//   SODG11_SSCC610_2403701_PLC/SODG11_SSCC610_2403701_PLC Instance <-> EtherCAT Master (EtherCAT)/IC02.T01 (EK1100)/IC02.T16 (EK1122)/Fix04.N13 (EP1008-0002)
//     Standard Inputs/Fix04.N13/I <-> Channel 1/Input
//     Standard Inputs/Fix04.N13/I @bit 1 <-> Channel 2/Input
//     Standard Inputs/Fix04.N13/I @bit 2 <-> Channel 3/Input
//     Standard Inputs/Fix04.N13/I @bit 3 <-> Channel 4/Input
//     Standard Inputs/Fix04.N13/I @bit 4 <-> Channel 5/Input
//     Standard Inputs/Fix04.N13/I @bit 5 <-> Channel 6/Input
//     Standard Inputs/Fix04.N13/I @bit 6 <-> Channel 7/Input
//     Standard Inputs/Fix04.N13/I @bit 7 <-> Channel 8/Input
//     Standard Inputs/Fix04.N13/InfoData/State <-> InfoData/State
//     Standard Inputs/Fix04.N13/Wc_State <-> WcState/WcState
//   SODG11_SSCC610_2403701_PLC/SODG11_SSCC610_2403701_PLC Instance <-> EtherCAT Master (EtherCAT)/IC02.T01 (EK1100)/IC02.T16 (EK1122)/Fix04.N14 (EP1008-0002)
//     Standard Inputs/Fix04.N14/I <-> Channel 1/Input
//     Standard Inputs/Fix04.N14/I @bit 1 <-> Channel 2/Input
//     Standard Inputs/Fix04.N14/I @bit 2 <-> Channel 3/Input
//     Standard Inputs/Fix04.N14/I @bit 3 <-> Channel 4/Input
//     Standard Inputs/Fix04.N14/I @bit 4 <-> Channel 5/Input
//     Standard Inputs/Fix04.N14/I @bit 5 <-> Channel 6/Input
//     Standard Inputs/Fix04.N14/I @bit 6 <-> Channel 7/Input
//     Standard Inputs/Fix04.N14/I @bit 7 <-> Channel 8/Input
//     Standard Inputs/Fix04.N14/InfoData/State <-> InfoData/State
//     Standard Inputs/Fix04.N14/Wc_State <-> WcState/WcState
//   SODG11_SSCC610_2403701_PLC/SODG11_SSCC610_2403701_PLC Instance <-> EtherCAT Master (EtherCAT)/IC02.T01 (EK1100)/IC02.T16 (EK1122)/Fix04.N15 (EP1008-0002)
//     Standard Inputs/Fix04.N15/I <-> Channel 1/Input
//     Standard Inputs/Fix04.N15/I @bit 1 <-> Channel 2/Input
//     Standard Inputs/Fix04.N15/I @bit 2 <-> Channel 3/Input
//     Standard Inputs/Fix04.N15/I @bit 3 <-> Channel 4/Input
//     Standard Inputs/Fix04.N15/I @bit 4 <-> Channel 5/Input
//     Standard Inputs/Fix04.N15/I @bit 5 <-> Channel 6/Input
//     Standard Inputs/Fix04.N15/I @bit 6 <-> Channel 7/Input
//     Standard Inputs/Fix04.N15/I @bit 7 <-> Channel 8/Input
//     Standard Inputs/Fix04.N15/InfoData/State <-> InfoData/State
//     Standard Inputs/Fix04.N15/Wc_State <-> WcState/WcState
//   SODG11_SSCC610_2403701_PLC/SODG11_SSCC610_2403701_PLC Instance <-> EtherCAT Master (EtherCAT)/IC02.T01 (EK1100)/IC02.T16 (EK1122)/Fix04.N16 (EP1008-0002)
//     Standard Inputs/Fix04.N16/I <-> Channel 1/Input
//     Standard Inputs/Fix04.N16/I @bit 1 <-> Channel 2/Input
//     Standard Inputs/Fix04.N16/I @bit 2 <-> Channel 3/Input
//     Standard Inputs/Fix04.N16/I @bit 3 <-> Channel 4/Input
//     Standard Inputs/Fix04.N16/I @bit 4 <-> Channel 5/Input
//     Standard Inputs/Fix04.N16/I @bit 5 <-> Channel 6/Input
//     Standard Inputs/Fix04.N16/I @bit 6 <-> Channel 7/Input
//     Standard Inputs/Fix04.N16/I @bit 7 <-> Channel 8/Input
//     Standard Inputs/Fix04.N16/InfoData/State <-> InfoData/State
//     Standard Inputs/Fix04.N16/Wc_State <-> WcState/WcState
//   SODG11_SSCC610_2403701_PLC/SODG11_SSCC610_2403701_PLC Instance <-> EtherCAT Master (EtherCAT)/IC02.T01 (EK1100)/IC02.T16 (EK1122)/Fix04.N17 (EP1008-0002)
//     Standard Inputs/Fix04.N17/I <-> Channel 1/Input
//     Standard Inputs/Fix04.N17/I @bit 1 <-> Channel 2/Input
//     Standard Inputs/Fix04.N17/I @bit 2 <-> Channel 3/Input
//     Standard Inputs/Fix04.N17/I @bit 3 <-> Channel 4/Input
//     Standard Inputs/Fix04.N17/I @bit 4 <-> Channel 5/Input
//     Standard Inputs/Fix04.N17/I @bit 5 <-> Channel 6/Input
//     Standard Inputs/Fix04.N17/I @bit 6 <-> Channel 7/Input
//     Standard Inputs/Fix04.N17/I @bit 7 <-> Channel 8/Input
//     Standard Inputs/Fix04.N17/InfoData/State <-> InfoData/State
//     Standard Inputs/Fix04.N17/Wc_State <-> WcState/WcState
//   SODG11_SSCC610_2403701_PLC/SODG11_SSCC610_2403701_PLC Instance <-> EtherCAT Master (EtherCAT)/IC02.T01 (EK1100)/IC02.T16 (EK1122)/Fix04.N18 (EP1008-0002)
//     Standard Inputs/Fix04.N18/I <-> Channel 1/Input
//     Standard Inputs/Fix04.N18/I @bit 1 <-> Channel 2/Input
//     Standard Inputs/Fix04.N18/I @bit 2 <-> Channel 3/Input
//     Standard Inputs/Fix04.N18/I @bit 3 <-> Channel 4/Input
//     Standard Inputs/Fix04.N18/I @bit 4 <-> Channel 5/Input
//     Standard Inputs/Fix04.N18/I @bit 5 <-> Channel 6/Input
//     Standard Inputs/Fix04.N18/I @bit 6 <-> Channel 7/Input
//     Standard Inputs/Fix04.N18/I @bit 7 <-> Channel 8/Input
//     Standard Inputs/Fix04.N18/InfoData/State <-> InfoData/State
//     Standard Inputs/Fix04.N18/Wc_State <-> WcState/WcState
//   SODG11_SSCC610_2403701_PLC/SODG11_SSCC610_2403701_PLC Instance <-> EtherCAT Master (EtherCAT)/IC02.T01 (EK1100)/IC02.T16 (EK1122)/Fix04.N19 (EP1008-0002)
//     Standard Inputs/Fix04.N19/I <-> Channel 1/Input
//     Standard Inputs/Fix04.N19/I @bit 1 <-> Channel 2/Input
//     Standard Inputs/Fix04.N19/I @bit 2 <-> Channel 3/Input
//     Standard Inputs/Fix04.N19/I @bit 3 <-> Channel 4/Input
//     Standard Inputs/Fix04.N19/I @bit 4 <-> Channel 5/Input
//     Standard Inputs/Fix04.N19/I @bit 5 <-> Channel 6/Input
//     Standard Inputs/Fix04.N19/I @bit 6 <-> Channel 7/Input
//     Standard Inputs/Fix04.N19/I @bit 7 <-> Channel 8/Input
//     Standard Inputs/Fix04.N19/InfoData/State <-> InfoData/State
//     Standard Inputs/Fix04.N19/Wc_State <-> WcState/WcState
//   SODG11_SSCC610_2403701_PLC/SODG11_SSCC610_2403701_PLC Instance <-> EtherCAT Master (EtherCAT)/IC02.T01 (EK1100)/IC02.T16 (EK1122)/Fix04.N20 (EP1008-0002)
//     Standard Inputs/Fix04.N20/I <-> Channel 1/Input
//     Standard Inputs/Fix04.N20/I @bit 1 <-> Channel 2/Input
//     Standard Inputs/Fix04.N20/I @bit 2 <-> Channel 3/Input
//     Standard Inputs/Fix04.N20/I @bit 3 <-> Channel 4/Input
//     Standard Inputs/Fix04.N20/I @bit 4 <-> Channel 5/Input
//     Standard Inputs/Fix04.N20/I @bit 5 <-> Channel 6/Input
//     Standard Inputs/Fix04.N20/I @bit 6 <-> Channel 7/Input
//     Standard Inputs/Fix04.N20/I @bit 7 <-> Channel 8/Input
//     Standard Inputs/Fix04.N20/InfoData/State <-> InfoData/State
//     Standard Inputs/Fix04.N20/Wc_State <-> WcState/WcState
//   SODG11_SSCC610_2403701_PLC/SODG11_SSCC610_2403701_PLC Instance <-> EtherCAT Master (EtherCAT)/IC02.T01 (EK1100)/IC02.T16 (EK1122)/Fix04.N21 (EP1008-0002)
//     Standard Inputs/Fix04.N21/I <-> Channel 1/Input
//     Standard Inputs/Fix04.N21/I @bit 1 <-> Channel 2/Input
//     Standard Inputs/Fix04.N21/I @bit 2 <-> Channel 3/Input
//     Standard Inputs/Fix04.N21/I @bit 3 <-> Channel 4/Input
//     Standard Inputs/Fix04.N21/I @bit 4 <-> Channel 5/Input
//     Standard Inputs/Fix04.N21/I @bit 5 <-> Channel 6/Input
//     Standard Inputs/Fix04.N21/I @bit 6 <-> Channel 7/Input
//     Standard Inputs/Fix04.N21/I @bit 7 <-> Channel 8/Input
//     Standard Inputs/Fix04.N21/InfoData/State <-> InfoData/State
//     Standard Inputs/Fix04.N21/Wc_State <-> WcState/WcState
//   SODG11_SSCC610_2403701_PLC/SODG11_SSCC610_2403701_PLC Instance <-> EtherCAT Master (EtherCAT)/IC02.T01 (EK1100)/IC02.T16 (EK1122)/Fix04.N22 (EP1008-0002)
//     Standard Inputs/Fix04.N22/I <-> Channel 1/Input
//     Standard Inputs/Fix04.N22/I @bit 1 <-> Channel 2/Input
//     Standard Inputs/Fix04.N22/I @bit 2 <-> Channel 3/Input
//     Standard Inputs/Fix04.N22/I @bit 3 <-> Channel 4/Input
//     Standard Inputs/Fix04.N22/I @bit 4 <-> Channel 5/Input
//     Standard Inputs/Fix04.N22/I @bit 5 <-> Channel 6/Input
//     Standard Inputs/Fix04.N22/I @bit 6 <-> Channel 7/Input
//     Standard Inputs/Fix04.N22/I @bit 7 <-> Channel 8/Input
//     Standard Inputs/Fix04.N22/InfoData/State <-> InfoData/State
//     Standard Inputs/Fix04.N22/Wc_State <-> WcState/WcState
//   SODG11_SSCC610_2403701_PLC/SODG11_SSCC610_2403701_PLC Instance <-> EtherCAT Master (EtherCAT)/IC02.T01 (EK1100)/IC02.T16 (EK1122)/Fix04.N90 (EP9214-0023)
//     Standard Inputs/Fix04.N90_STAT/Channel_1/Channel_Error <-> DPO Inputs Channel 1/Channel Error
//     Standard Inputs/Fix04.N90_STAT/Channel_2/Channel_Error <-> DPO Inputs Channel 2/Channel Error
//     Standard Inputs/Fix04.N90_STAT/Channel_3/Channel_Error <-> DPO Inputs Channel 3/Channel Error
